LIN {X 0,Y 252.617,Z 375.024,A -85,B 0,C 180,E1 -18754.516,E2 -18754.516} C_VEL
LIN {X 0,Y 250.193,Z 375.321,A -85,B 0,C 180,E1 -18756.259,E2 -18756.259} C_VEL
LIN {X 0,Y 249.15,Z 375.448,A -85,B 0,C 180,E1 -18757.61,E2 -18757.61} C_VEL
LIN {X 0,Y 249.065,Z 375.457,A -85,B 0,C 180,E1 -18758.068,E2 -18758.068} C_VEL
LIN {X 0,Y 249.093,Z 375.454,A -85,B 0,C 180,E1 -18760.461,E2 -18760.461} C_VEL
LIN {X 0,Y 249.089,Z 375.456,A -85,B 0,C 180,E1 -18762.815,E2 -18762.815} C_VEL
LIN {X 0,Y 249.094,Z 375.457,A -85,B 0,C 180,E1 -18767.382,E2 -18767.382} C_VEL
LIN {X 0,Y 249.049,Z 375.461,A -85,B 0,C 180,E1 -18771.626,E2 -18771.626} C_VEL
LIN {X 0,Y 249.193,Z 375.539,A -85,B 0,C 180,E1 -18775.523,E2 -18775.523} C_VEL
LIN {X 0,Y 252.491,Z 392.1,A -85,B 0,C 180,E1 -18780.852,E2 -18780.852} C_VEL
LIN {X 0,Y 253.054,Z 396.272,A -85,B 0,C 180,E1 -18782.147,E2 -18782.147} C_VEL
LIN {X 0,Y 251.958,Z 403.5,A -85,B 0,C 180,E1 -18784.275,E2 -18784.275} C_VEL
LIN {X 0,Y 252.886,Z 424.337,A -85,B 0,C 180,E1 -18785.283,E2 -18785.283} C_VEL
LIN {X 0,Y 255.604,Z 456.086,A -85,B 0,C 180,E1 -18786.853,E2 -18786.853} C_VEL
LIN {X 0,Y 253.392,Z 514.144,A -85,B 0,C 180,E1 -18789.558,E2 -18789.558} C_VEL
LIN {X 0,Y 252.579,Z 527.545,A -85,B 0,C 180,E1 -18790.496,E2 -18790.496} C_VEL
LIN {X 0,Y 251.524,Z 541.094,A -85,B 0,C 180,E1 -18791.809,E2 -18791.809} C_VEL
LIN {X 0,Y 250.583,Z 553.006,A -85,B 0,C 180,E1 -18793.298,E2 -18793.298} C_VEL
LIN {X 0,Y 249.728,Z 563.328,A -85,B 0,C 180,E1 -18794.913,E2 -18794.913} C_VEL
LIN {X 0,Y 248.987,Z 573.942,A -85,B 0,C 180,E1 -18796.951,E2 -18796.951} C_VEL
LIN {X 0,Y 248.46,Z 582.589,A -85,B 0,C 180,E1 -18798.995,E2 -18798.995} C_VEL
LIN {X 0,Y 248.115,Z 590.984,A -85,B 0,C 180,E1 -18801.45,E2 -18801.45} C_VEL
LIN {X 0,Y 248.097,Z 596.674,A -85,B 0,C 180,E1 -18803.496,E2 -18803.496} C_VEL
LIN {X 0,Y 248.11,Z 602.079,A -85,B 0,C 180,E1 -18805.941,E2 -18805.941} C_VEL
LIN {X 0,Y 248.161,Z 606.143,A -85,B 0,C 180,E1 -18808.379,E2 -18808.379} C_VEL
LIN {X 0,Y 248.142,Z 608.182,A -85,B 0,C 180,E1 -18810.002,E2 -18810.002} C_VEL
LIN {X 0,Y 247.812,Z 609.634,A -85,B 0,C 180,E1 -18811.627,E2 -18811.627} C_VEL
LIN {X 0,Y 247.537,Z 610.654,A -85,B 0,C 180,E1 -18813.257,E2 -18813.257} C_VEL
LIN {X 0,Y 247.286,Z 611.402,A -85,B 0,C 180,E1 -18815.888,E2 -18815.888} C_VEL
LIN {X 0,Y 247.279,Z 611.195,A -85,B 0,C 180,E1 -18818.172,E2 -18818.172} C_VEL
LIN {X 0,Y 247.949,Z 609.525,A -85,B 0,C 180,E1 -18821.446,E2 -18821.446} C_VEL
LIN {X 0,Y 248.585,Z 608.119,A -85,B 0,C 180,E1 -18823.074,E2 -18823.074} C_VEL
LIN {X 0,Y 250.166,Z 605.234,A -85,B 0,C 180,E1 -18825.481,E2 -18825.481} C_VEL
LIN {X 0,Y 252.071,Z 601.416,A -85,B 0,C 180,E1 -18827.862,E2 -18827.862} C_VEL
LIN {X 0,Y 254.472,Z 596.794,A -85,B 0,C 180,E1 -18830.113,E2 -18830.113} C_VEL
LIN {X 0,Y 258.315,Z 589.612,A -85,B 0,C 180,E1 -18832.813,E2 -18832.813} C_VEL
LIN {X 0,Y 262.794,Z 580.873,A -85,B 0,C 180,E1 -18835.336,E2 -18835.336} C_VEL
LIN {X 0,Y 267.178,Z 571.753,A -85,B 0,C 180,E1 -18837.41,E2 -18837.41} C_VEL
LIN {X 0,Y 271.297,Z 562.717,A -85,B 0,C 180,E1 -18839.061,E2 -18839.061} C_VEL
LIN {X 0,Y 275.703,Z 552.071,A -85,B 0,C 180,E1 -18840.654,E2 -18840.654} C_VEL
LIN {X 0,Y 280.786,Z 538.915,A -85,B 0,C 180,E1 -18842.134,E2 -18842.134} C_VEL
LIN {X 0,Y 285.07,Z 525.941,A -85,B 0,C 180,E1 -18843.269,E2 -18843.269} C_VEL
LIN {X 0,Y 289,Z 511.6,A -85,B 0,C 180,E1 -18844.243,E2 -18844.243} C_VEL
LIN {X 0,Y 292.448,Z 494.65,A -85,B 0,C 180,E1 -18845.109,E2 -18845.109} C_VEL
LIN {X 0,Y 297.197,Z 467.184,A -85,B 0,C 180,E1 -18846.361,E2 -18846.361} C_VEL
LIN {X 0,Y 297.851,Z 457.621,A -85,B 0,C 180,E1 -18847.315,E2 -18847.315} C_VEL
LIN {X 0,Y 297.997,Z 452.789,A -85,B 0,C 180,E1 -18847.929,E2 -18847.929} C_VEL
LIN {X 0,Y 296.629,Z 446.766,A -85,B 0,C 180,E1 -18849.823,E2 -18849.823} C_VEL
LIN {X 0,Y 295.412,Z 441.538,A -85,B 0,C 180,E1 -18852.263,E2 -18852.263} C_VEL
LIN {X 0,Y 294.804,Z 438.826,A -85,B 0,C 180,E1 -18854.79,E2 -18854.79} C_VEL
LIN {X 0,Y 295.112,Z 437.625,A -85,B 0,C 180,E1 -18856.988,E2 -18856.988} C_VEL
LIN {X 0,Y 295.976,Z 437.721,A -85,B 0,C 180,E1 -18858.968,E2 -18858.968} C_VEL
LIN {X 0,Y 297.649,Z 439.646,A -85,B 0,C 180,E1 -18861.321,E2 -18861.321} C_VEL
LIN {X 0,Y 299.387,Z 442.577,A -85,B 0,C 180,E1 -18863.094,E2 -18863.094} C_VEL
LIN {X 0,Y 300.465,Z 444.609,A -85,B 0,C 180,E1 -18864.024,E2 -18864.024} C_VEL
LIN {X 0,Y 293.198,Z 484.481,A -85,B 0,C 180,E1 -18865.871,E2 -18865.871} C_VEL
LIN {X 0,Y 290.285,Z 498.234,A -85,B 0,C 180,E1 -18866.786,E2 -18866.786} C_VEL
LIN {X 0,Y 287.106,Z 510.262,A -85,B 0,C 180,E1 -18867.831,E2 -18867.831} C_VEL
LIN {X 0,Y 282.774,Z 523.775,A -85,B 0,C 180,E1 -18869.369,E2 -18869.369} C_VEL
LIN {X 0,Y 278.638,Z 534.629,A -85,B 0,C 180,E1 -18870.952,E2 -18870.952} C_VEL
LIN {X 0,Y 273.95,Z 545.313,A -85,B 0,C 180,E1 -18872.911,E2 -18872.911} C_VEL
LIN {X 0,Y 269.585,Z 553.981,A -85,B 0,C 180,E1 -18874.936,E2 -18874.936} C_VEL
LIN {X 0,Y 265.689,Z 561.042,A -85,B 0,C 180,E1 -18877.035,E2 -18877.035} C_VEL
LIN {X 0,Y 261.627,Z 567.566,A -85,B 0,C 180,E1 -18879.56,E2 -18879.56} C_VEL
LIN {X 0,Y 258.489,Z 571.94,A -85,B 0,C 180,E1 -18881.78,E2 -18881.78} C_VEL
LIN {X 0,Y 255.829,Z 575.254,A -85,B 0,C 180,E1 -18884.055,E2 -18884.055} C_VEL
LIN {X 0,Y 252.829,Z 578.178,A -85,B 0,C 180,E1 -18887.151,E2 -18887.151} C_VEL
LIN {X 0,Y 251.574,Z 579.01,A -85,B 0,C 180,E1 -18888.723,E2 -18888.723} C_VEL
LIN {X 0,Y 250.49,Z 579.42,A -85,B 0,C 180,E1 -18890.308,E2 -18890.308} C_VEL
LIN {X 0,Y 249.649,Z 579.428,A -85,B 0,C 180,E1 -18891.908,E2 -18891.908} C_VEL
LIN {X 0,Y 249.079,Z 579.037,A -85,B 0,C 180,E1 -18893.519,E2 -18893.519} C_VEL
LIN {X 0,Y 248.577,Z 578.237,A -85,B 0,C 180,E1 -18895.134,E2 -18895.134} C_VEL
LIN {X 0,Y 248.045,Z 577.007,A -85,B 0,C 180,E1 -18896.751,E2 -18896.751} C_VEL
LIN {X 0,Y 247.507,Z 574.382,A -85,B 0,C 180,E1 -18899.186,E2 -18899.186} C_VEL
LIN {X 0,Y 247.375,Z 570.743,A -85,B 0,C 180,E1 -18901.628,E2 -18901.628} C_VEL
LIN {X 0,Y 247.57,Z 565.989,A -85,B 0,C 180,E1 -18904.07,E2 -18904.07} C_VEL
LIN {X 0,Y 247.729,Z 559.198,A -85,B 0,C 180,E1 -18906.801,E2 -18906.801} C_VEL
LIN {X 0,Y 248.148,Z 552.516,A -85,B 0,C 180,E1 -18908.961,E2 -18908.961} C_VEL
LIN {X 0,Y 248.804,Z 543.249,A -85,B 0,C 180,E1 -18911.404,E2 -18911.404} C_VEL
LIN {X 0,Y 249.629,Z 532.822,A -85,B 0,C 180,E1 -18913.638,E2 -18913.638} C_VEL
LIN {X 0,Y 250.547,Z 522.317,A -85,B 0,C 180,E1 -18915.455,E2 -18915.455} C_VEL
LIN {X 0,Y 251.572,Z 509.36,A -85,B 0,C 180,E1 -18917.267,E2 -18917.267} C_VEL
LIN {X 0,Y 252.418,Z 495.882,A -85,B 0,C 180,E1 -18918.726,E2 -18918.726} C_VEL
LIN {X 0,Y 253.216,Z 482.499,A -85,B 0,C 180,E1 -18919.824,E2 -18919.824} C_VEL
LIN {X 0,Y 253.806,Z 467.784,A -85,B 0,C 180,E1 -18920.674,E2 -18920.674} C_VEL
LIN {X 0,Y 256.435,Z 400.26,A -85,B 0,C 180,E1 -18923.69,E2 -18923.69} C_VEL
LIN {X 0,Y 249.152,Z 375.446,A -85,B 0,C 180,E1 -18925.17,E2 -18925.17} C_VEL
LIN {X 0,Y 249.09,Z 375.455,A -85,B 0,C 180,E1 -18928.993,E2 -18928.993} C_VEL
LIN {X 0,Y 249.039,Z 375.462,A -85,B 0,C 180,E1 -18932.424,E2 -18932.424} C_VEL
LIN {X 0,Y 249.064,Z 375.463,A -85,B 0,C 180,E1 -18936.34,E2 -18936.34} C_VEL
LIN {X 0,Y 249.011,Z 375.465,A -85,B 0,C 180,E1 -18940.477,E2 -18940.477} C_VEL
LIN {X 0,Y 249.007,Z 375.466,A -85,B 0,C 180,E1 -18944.878,E2 -18944.878} C_VEL
LIN {X 0,Y 249.021,Z 375.463,A -85,B 0,C 180,E1 -18947.362,E2 -18947.362} C_VEL
LIN {X 0,Y 249.053,Z 375.462,A -85,B 0,C 180,E1 -18952.197,E2 -18952.197} C_VEL
LIN {X 0,Y 249.063,Z 375.459,A -85,B 0,C 180,E1 -18955.64,E2 -18955.64} C_VEL
LIN {X 0,Y 249.055,Z 375.457,A -85,B 0,C 180,E1 -18959.472,E2 -18959.472} C_VEL
LIN {X 0,Y 249.076,Z 375.457,A -85,B 0,C 180,E1 -18963.161,E2 -18963.161} C_VEL
LIN {X 0,Y 249.083,Z 375.455,A -85,B 0,C 180,E1 -18966.731,E2 -18966.731} C_VEL
LIN {X 0,Y 249.115,Z 375.455,A -85,B 0,C 180,E1 -18970.21,E2 -18970.21} C_VEL
LIN {X 0,Y 249.245,Z 375.437,A -85,B 0,C 180,E1 -18973.62,E2 -18973.62} C_VEL
LIN {X 0,Y 249.247,Z 375.436,A -85,B 0,C 180,E1 -18978.615,E2 -18978.615} C_VEL
LIN {X 0,Y 249.457,Z 375.413,A -85,B 0,C 180,E1 -18981.9,E2 -18981.9} C_VEL
LIN {X 0,Y 249.3,Z 375.427,A -85,B 0,C 180,E1 -18985.147,E2 -18985.147} C_VEL
LIN {X 0,Y 249.678,Z 375.383,A -85,B 0,C 180,E1 -18988.385,E2 -18988.385} C_VEL
LIN {X 0,Y 249.678,Z 375.383,A -85,B 0,C 180,E1 -18991.611,E2 -18991.611} C_VEL
LIN {X 0,Y 249.463,Z 375.409,A -85,B 0,C 180,E1 -18996.468,E2 -18996.468} C_VEL
LIN {X 0,Y 249.424,Z 375.416,A -85,B 0,C 180,E1 -18999.731,E2 -18999.731} C_VEL
LIN {X 0,Y 249.205,Z 375.44,A -85,B 0,C 180,E1 -19004.701,E2 -19004.701} C_VEL
LIN {X 0,Y 249.138,Z 375.452,A -85,B 0,C 180,E1 -19008.075,E2 -19008.075} C_VEL
LIN {X 0,Y 249.085,Z 375.456,A -85,B 0,C 180,E1 -19011.516,E2 -19011.516} C_VEL
LIN {X 0,Y 249.128,Z 375.452,A -85,B 0,C 180,E1 -19015.48,E2 -19015.48} C_VEL
LIN {X 0,Y 249.077,Z 375.456,A -85,B 0,C 180,E1 -19018.99,E2 -19018.99} C_VEL
LIN {X 0,Y 249.032,Z 375.462,A -85,B 0,C 180,E1 -19022.423,E2 -19022.423} C_VEL
LIN {X 0,Y 249.071,Z 375.458,A -85,B 0,C 180,E1 -19026.336,E2 -19026.336} C_VEL
LIN {X 0,Y 249.076,Z 375.456,A -85,B 0,C 180,E1 -19030.461,E2 -19030.461} C_VEL
LIN {X 0,Y 249.082,Z 375.456,A -85,B 0,C 180,E1 -19032.81,E2 -19032.81} C_VEL
LIN {X 0,Y 249.093,Z 375.455,A -85,B 0,C 180,E1 -19037.379,E2 -19037.379} C_VEL
LIN {X 0,Y 249.046,Z 375.464,A -85,B 0,C 180,E1 -19041.623,E2 -19041.623} C_VEL
LIN {X 0,Y 249.054,Z 375.462,A -85,B 0,C 180,E1 -19045.641,E2 -19045.641} C_VEL
LIN {X 0,Y 249.045,Z 375.462,A -85,B 0,C 180,E1 -19049.472,E2 -19049.472} C_VEL
LIN {X 0,Y 249.068,Z 375.459,A -85,B 0,C 180,E1 -19053.162,E2 -19053.162} C_VEL
LIN {X 0,Y 249.071,Z 375.455,A -85,B 0,C 180,E1 -19056.732,E2 -19056.732} C_VEL
LIN {X 0,Y 249.102,Z 375.454,A -85,B 0,C 180,E1 -19060.211,E2 -19060.211} C_VEL
LIN {X 0,Y 249.233,Z 375.439,A -85,B 0,C 180,E1 -19063.621,E2 -19063.621} C_VEL
LIN {X 0,Y 249.244,Z 375.436,A -85,B 0,C 180,E1 -19068.616,E2 -19068.616} C_VEL
LIN {X 0,Y 249.475,Z 375.407,A -85,B 0,C 180,E1 -19071.903,E2 -19071.903} C_VEL
LIN {X 0,Y 249.433,Z 375.412,A -85,B 0,C 180,E1 -19076.77,E2 -19076.77} C_VEL
LIN {X 0,Y 249.727,Z 375.376,A -85,B 0,C 180,E1 -19080,E2 -19080} C_VEL
LIN {X 0,Y 249.431,Z 375.413,A -85,B 0,C 180,E1 -19083.231,E2 -19083.231} C_VEL
LIN {X 0,Y 249.476,Z 375.407,A -85,B 0,C 180,E1 -19088.098,E2 -19088.098} C_VEL
LIN {X 0,Y 249.245,Z 375.437,A -85,B 0,C 180,E1 -19091.384,E2 -19091.384} C_VEL
LIN {X 0,Y 249.234,Z 375.437,A -85,B 0,C 180,E1 -19096.379,E2 -19096.379} C_VEL
LIN {X 0,Y 249.079,Z 375.459,A -85,B 0,C 180,E1 -19101.519,E2 -19101.519} C_VEL
LIN {X 0,Y 249.122,Z 375.454,A -85,B 0,C 180,E1 -19105.483,E2 -19105.483} C_VEL
LIN {X 0,Y 249.065,Z 375.457,A -85,B 0,C 180,E1 -19108.99,E2 -19108.99} C_VEL
LIN {X 0,Y 249.029,Z 375.463,A -85,B 0,C 180,E1 -19112.426,E2 -19112.426} C_VEL
LIN {X 0,Y 249.069,Z 375.456,A -85,B 0,C 180,E1 -19116.339,E2 -19116.339} C_VEL
LIN {X 0,Y 249.065,Z 375.457,A -85,B 0,C 180,E1 -19118.068,E2 -19118.068} C_VEL
LIN {X 0,Y 248.389,Z 375.545,A -85,B 0,C 180,E1 -19119.418,E2 -19119.418} C_VEL
LIN {X 0,Y 245.511,Z 375.903,A -85,B 0,C 180,E1 -19121.617,E2 -19121.617} C_VEL
LIN {X 0,Y 243.082,Z 376.206,A -85,B 0,C 180,E1 -19123.409,E2 -19123.409} C_VEL
LIN {X 0,Y 242.058,Z 376.331,A -85,B 0,C 180,E1 -19124.8,E2 -19124.8} C_VEL
LIN {X 0,Y 241.985,Z 376.336,A -85,B 0,C 180,E1 -19125.271,E2 -19125.271} C_VEL
LIN {X 0,Y 242.006,Z 376.339,A -85,B 0,C 180,E1 -19129.031,E2 -19129.031} C_VEL
LIN {X 0,Y 242.012,Z 376.336,A -85,B 0,C 180,E1 -19132.425,E2 -19132.425} C_VEL
LIN {X 0,Y 242.159,Z 376.504,A -85,B 0,C 180,E1 -19135.409,E2 -19135.409} C_VEL
LIN {X 0,Y 245.444,Z 392.998,A -85,B 0,C 180,E1 -19140.874,E2 -19140.874} C_VEL
LIN {X 0,Y 246.019,Z 395.864,A -85,B 0,C 180,E1 -19141.796,E2 -19141.796} C_VEL
LIN {X 0,Y 244.986,Z 402.846,A -85,B 0,C 180,E1 -19143.945,E2 -19143.945} C_VEL
LIN {X 0,Y 245.82,Z 424.179,A -85,B 0,C 180,E1 -19145.029,E2 -19145.029} C_VEL
LIN {X 0,Y 248.539,Z 456.485,A -85,B 0,C 180,E1 -19146.681,E2 -19146.681} C_VEL
LIN {X 0,Y 246.337,Z 513.372,A -85,B 0,C 180,E1 -19149.437,E2 -19149.437} C_VEL
LIN {X 0,Y 245.574,Z 526.114,A -85,B 0,C 180,E1 -19150.353,E2 -19150.353} C_VEL
LIN {X 0,Y 244.596,Z 538.728,A -85,B 0,C 180,E1 -19151.577,E2 -19151.577} C_VEL
LIN {X 0,Y 243.581,Z 551.828,A -85,B 0,C 180,E1 -19153.232,E2 -19153.232} C_VEL
LIN {X 0,Y 242.707,Z 562.251,A -85,B 0,C 180,E1 -19154.896,E2 -19154.896} C_VEL
LIN {X 0,Y 241.955,Z 572.94,A -85,B 0,C 180,E1 -19156.993,E2 -19156.993} C_VEL
LIN {X 0,Y 241.439,Z 581.655,A -85,B 0,C 180,E1 -19159.096,E2 -19159.096} C_VEL
LIN {X 0,Y 241.112,Z 590.081,A -85,B 0,C 180,E1 -19161.622,E2 -19161.622} C_VEL
LIN {X 0,Y 241.112,Z 596.823,A -85,B 0,C 180,E1 -19164.147,E2 -19164.147} C_VEL
LIN {X 0,Y 241.115,Z 602.029,A -85,B 0,C 180,E1 -19166.66,E2 -19166.66} C_VEL
LIN {X 0,Y 241.167,Z 605.897,A -85,B 0,C 180,E1 -19169.167,E2 -19169.167} C_VEL
LIN {X 0,Y 240.793,Z 608.515,A -85,B 0,C 180,E1 -19171.674,E2 -19171.674} C_VEL
LIN {X 0,Y 240.494,Z 609.654,A -85,B 0,C 180,E1 -19173.353,E2 -19173.353} C_VEL
LIN {X 0,Y 240.23,Z 610.594,A -85,B 0,C 180,E1 -19175.909,E2 -19175.909} C_VEL
LIN {X 0,Y 240.232,Z 610.572,A -85,B 0,C 180,E1 -19178.413,E2 -19178.413} C_VEL
LIN {X 0,Y 240.48,Z 610.095,A -85,B 0,C 180,E1 -19180.101,E2 -19180.101} C_VEL
LIN {X 0,Y 241.647,Z 607.937,A -85,B 0,C 180,E1 -19183.456,E2 -19183.456} C_VEL
LIN {X 0,Y 243.954,Z 604.238,A -85,B 0,C 180,E1 -19186.745,E2 -19186.745} C_VEL
LIN {X 0,Y 246.1,Z 600.387,A -85,B 0,C 180,E1 -19189.174,E2 -19189.174} C_VEL
LIN {X 0,Y 249.066,Z 595.535,A -85,B 0,C 180,E1 -19191.522,E2 -19191.522} C_VEL
LIN {X 0,Y 252.521,Z 589.616,A -85,B 0,C 180,E1 -19193.802,E2 -19193.802} C_VEL
LIN {X 0,Y 257.239,Z 581.183,A -85,B 0,C 180,E1 -19196.359,E2 -19196.359} C_VEL
LIN {X 0,Y 261.893,Z 572.344,A -85,B 0,C 180,E1 -19198.448,E2 -19198.448} C_VEL
LIN {X 0,Y 267.118,Z 561.712,A -85,B 0,C 180,E1 -19200.431,E2 -19200.431} C_VEL
LIN {X 0,Y 271.888,Z 551.1,A -85,B 0,C 180,E1 -19202.001,E2 -19202.001} C_VEL
LIN {X 0,Y 277.23,Z 538.071,A -85,B 0,C 180,E1 -19203.463,E2 -19203.463} C_VEL
LIN {X 0,Y 281.752,Z 525.166,A -85,B 0,C 180,E1 -19204.59,E2 -19204.59} C_VEL
LIN {X 0,Y 286.049,Z 510.245,A -85,B 0,C 180,E1 -19205.597,E2 -19205.597} C_VEL
LIN {X 0,Y 289.59,Z 494.129,A -85,B 0,C 180,E1 -19206.413,E2 -19206.413} C_VEL
LIN {X 0,Y 294.264,Z 468.85,A -85,B 0,C 180,E1 -19207.571,E2 -19207.571} C_VEL
LIN {X 0,Y 295.084,Z 459.535,A -85,B 0,C 180,E1 -19208.557,E2 -19208.557} C_VEL
LIN {X 0,Y 295.153,Z 457.377,A -85,B 0,C 180,E1 -19208.873,E2 -19208.873} C_VEL
LIN {X 0,Y 294.254,Z 452.71,A -85,B 0,C 180,E1 -19210.44,E2 -19210.44} C_VEL
LIN {X 0,Y 293.345,Z 447.937,A -85,B 0,C 180,E1 -19212.734,E2 -19212.734} C_VEL
LIN {X 0,Y 292.987,Z 445.294,A -85,B 0,C 180,E1 -19215.375,E2 -19215.375} C_VEL
LIN {X 0,Y 293.243,Z 444.54,A -85,B 0,C 180,E1 -19216.832,E2 -19216.832} C_VEL
LIN {X 0,Y 294.16,Z 444.64,A -85,B 0,C 180,E1 -19219.006,E2 -19219.006} C_VEL
LIN {X 0,Y 295.622,Z 446.463,A -85,B 0,C 180,E1 -19221.145,E2 -19221.145} C_VEL
LIN {X 0,Y 297.241,Z 449.345,A -85,B 0,C 180,E1 -19222.901,E2 -19222.901} C_VEL
LIN {X 0,Y 289.709,Z 488.112,A -85,B 0,C 180,E1 -19224.766,E2 -19224.766} C_VEL
LIN {X 0,Y 286.648,Z 501.036,A -85,B 0,C 180,E1 -19225.673,E2 -19225.673} C_VEL
LIN {X 0,Y 282.835,Z 513.919,A -85,B 0,C 180,E1 -19226.861,E2 -19226.861} C_VEL
LIN {X 0,Y 278.725,Z 525.572,A -85,B 0,C 180,E1 -19228.24,E2 -19228.24} C_VEL
LIN {X 0,Y 273.913,Z 537.133,A -85,B 0,C 180,E1 -19229.978,E2 -19229.978} C_VEL
LIN {X 0,Y 268.966,Z 547.375,A -85,B 0,C 180,E1 -19231.944,E2 -19231.944} C_VEL
LIN {X 0,Y 264.338,Z 555.79,A -85,B 0,C 180,E1 -19233.979,E2 -19233.979} C_VEL
LIN {X 0,Y 260.171,Z 562.604,A -85,B 0,C 180,E1 -19236.096,E2 -19236.096} C_VEL
LIN {X 0,Y 256.415,Z 568.11,A -85,B 0,C 180,E1 -19238.283,E2 -19238.283} C_VEL
LIN {X 0,Y 253.046,Z 572.496,A -85,B 0,C 180,E1 -19240.532,E2 -19240.532} C_VEL
LIN {X 0,Y 249.99,Z 575.942,A -85,B 0,C 180,E1 -19242.915,E2 -19242.915} C_VEL
LIN {X 0,Y 247.564,Z 578.23,A -85,B 0,C 180,E1 -19245.197,E2 -19245.197} C_VEL
LIN {X 0,Y 244.69,Z 579.952,A -85,B 0,C 180,E1 -19248.401,E2 -19248.401} C_VEL
LIN {X 0,Y 243.539,Z 580.227,A -85,B 0,C 180,E1 -19250.029,E2 -19250.029} C_VEL
LIN {X 0,Y 242.649,Z 580.085,A -85,B 0,C 180,E1 -19251.673,E2 -19251.673} C_VEL
LIN {X 0,Y 241.507,Z 578.539,A -85,B 0,C 180,E1 -19254.991,E2 -19254.991} C_VEL
LIN {X 0,Y 240.961,Z 577.184,A -85,B 0,C 180,E1 -19256.656,E2 -19256.656} C_VEL
LIN {X 0,Y 240.419,Z 574.323,A -85,B 0,C 180,E1 -19259.162,E2 -19259.162} C_VEL
LIN {X 0,Y 240.296,Z 570.436,A -85,B 0,C 180,E1 -19261.676,E2 -19261.676} C_VEL
LIN {X 0,Y 240.504,Z 565.439,A -85,B 0,C 180,E1 -19264.189,E2 -19264.189} C_VEL
LIN {X 0,Y 240.648,Z 558.892,A -85,B 0,C 180,E1 -19266.793,E2 -19266.793} C_VEL
LIN {X 0,Y 241.125,Z 551.302,A -85,B 0,C 180,E1 -19269.225,E2 -19269.225} C_VEL
LIN {X 0,Y 241.823,Z 541.678,A -85,B 0,C 180,E1 -19271.738,E2 -19271.738} C_VEL
LIN {X 0,Y 242.735,Z 530.669,A -85,B 0,C 180,E1 -19274.033,E2 -19274.033} C_VEL
LIN {X 0,Y 243.651,Z 519.657,A -85,B 0,C 180,E1 -19275.904,E2 -19275.904} C_VEL
LIN {X 0,Y 244.58,Z 507.492,A -85,B 0,C 180,E1 -19277.561,E2 -19277.561} C_VEL
LIN {X 0,Y 245.457,Z 493.991,A -85,B 0,C 180,E1 -19279.008,E2 -19279.008} C_VEL
LIN {X 0,Y 246.327,Z 479.034,A -85,B 0,C 180,E1 -19280.185,E2 -19280.185} C_VEL
LIN {X 0,Y 247.021,Z 460.314,A -85,B 0,C 180,E1 -19281.16,E2 -19281.16} C_VEL
LIN {X 0,Y 249.366,Z 401.443,A -85,B 0,C 180,E1 -19283.907,E2 -19283.907} C_VEL
LIN {X 0,Y 242.104,Z 376.324,A -85,B 0,C 180,E1 -19285.457,E2 -19285.457} C_VEL
LIN {X 0,Y 242.036,Z 376.334,A -85,B 0,C 180,E1 -19289.579,E2 -19289.579} C_VEL
LIN {X 0,Y 241.994,Z 376.336,A -85,B 0,C 180,E1 -19293.49,E2 -19293.49} C_VEL
LIN {X 0,Y 241.997,Z 376.339,A -85,B 0,C 180,E1 -19297.58,E2 -19297.58} C_VEL
LIN {X 0,Y 241.943,Z 376.345,A -85,B 0,C 180,E1 -19301.921,E2 -19301.921} C_VEL
LIN {X 0,Y 241.939,Z 376.348,A -85,B 0,C 180,E1 -19306.57,E2 -19306.57} C_VEL
LIN {X 0,Y 241.962,Z 376.344,A -85,B 0,C 180,E1 -19310.28,E2 -19310.28} C_VEL
LIN {X 0,Y 242.041,Z 376.335,A -85,B 0,C 180,E1 -19314.496,E2 -19314.496} C_VEL
LIN {X 0,Y 241.979,Z 376.34,A -85,B 0,C 180,E1 -19318.479,E2 -19318.479} C_VEL
LIN {X 0,Y 242.011,Z 376.34,A -85,B 0,C 180,E1 -19322.311,E2 -19322.311} C_VEL
LIN {X 0,Y 242.061,Z 376.334,A -85,B 0,C 180,E1 -19326.014,E2 -19326.014} C_VEL
LIN {X 0,Y 242.041,Z 376.332,A -85,B 0,C 180,E1 -19329.606,E2 -19329.606} C_VEL
LIN {X 0,Y 242.166,Z 376.318,A -85,B 0,C 180,E1 -19333.277,E2 -19333.277} C_VEL
LIN {X 0,Y 242.184,Z 376.317,A -85,B 0,C 180,E1 -19338.278,E2 -19338.278} C_VEL
LIN {X 0,Y 242.403,Z 376.29,A -85,B 0,C 180,E1 -19341.663,E2 -19341.663} C_VEL
LIN {X 0,Y 242.261,Z 376.303,A -85,B 0,C 180,E1 -19345.005,E2 -19345.005} C_VEL
LIN {X 0,Y 242.639,Z 376.261,A -85,B 0,C 180,E1 -19348.338,E2 -19348.338} C_VEL
LIN {X 0,Y 242.638,Z 376.261,A -85,B 0,C 180,E1 -19351.658,E2 -19351.658} C_VEL
LIN {X 0,Y 242.435,Z 376.284,A -85,B 0,C 180,E1 -19356.657,E2 -19356.657} C_VEL
LIN {X 0,Y 242.345,Z 376.298,A -85,B 0,C 180,E1 -19360.018,E2 -19360.018} C_VEL
LIN {X 0,Y 242.166,Z 376.317,A -85,B 0,C 180,E1 -19365.139,E2 -19365.139} C_VEL
LIN {X 0,Y 242.072,Z 376.329,A -85,B 0,C 180,E1 -19368.622,E2 -19368.622} C_VEL
LIN {X 0,Y 242.01,Z 376.337,A -85,B 0,C 180,E1 -19372.178,E2 -19372.178} C_VEL
LIN {X 0,Y 242.063,Z 376.334,A -85,B 0,C 180,E1 -19375.836,E2 -19375.836} C_VEL
LIN {X 0,Y 242.025,Z 376.336,A -85,B 0,C 180,E1 -19379.578,E2 -19379.578} C_VEL
LIN {X 0,Y 241.987,Z 376.341,A -85,B 0,C 180,E1 -19383.489,E2 -19383.489} C_VEL
LIN {X 0,Y 242.008,Z 376.339,A -85,B 0,C 180,E1 -19387.576,E2 -19387.576} C_VEL
LIN {X 0,Y 242.026,Z 376.338,A -85,B 0,C 180,E1 -19391.9,E2 -19391.9} C_VEL
LIN {X 0,Y 242.019,Z 376.335,A -85,B 0,C 180,E1 -19396.547,E2 -19396.547} C_VEL
LIN {X 0,Y 242.004,Z 376.338,A -85,B 0,C 180,E1 -19400.29,E2 -19400.29} C_VEL
LIN {X 0,Y 242.029,Z 376.334,A -85,B 0,C 180,E1 -19404.496,E2 -19404.496} C_VEL
LIN {X 0,Y 241.969,Z 376.341,A -85,B 0,C 180,E1 -19408.479,E2 -19408.479} C_VEL
LIN {X 0,Y 242.004,Z 376.338,A -85,B 0,C 180,E1 -19412.312,E2 -19412.312} C_VEL
LIN {X 0,Y 242.049,Z 376.332,A -85,B 0,C 180,E1 -19416.015,E2 -19416.015} C_VEL
LIN {X 0,Y 242.029,Z 376.339,A -85,B 0,C 180,E1 -19419.607,E2 -19419.607} C_VEL
LIN {X 0,Y 242.154,Z 376.32,A -85,B 0,C 180,E1 -19423.278,E2 -19423.278} C_VEL
LIN {X 0,Y 242.178,Z 376.316,A -85,B 0,C 180,E1 -19428.28,E2 -19428.28} C_VEL
LIN {X 0,Y 242.426,Z 376.287,A -85,B 0,C 180,E1 -19431.666,E2 -19431.666} C_VEL
LIN {X 0,Y 242.254,Z 376.306,A -85,B 0,C 180,E1 -19435.007,E2 -19435.007} C_VEL
LIN {X 0,Y 242.631,Z 376.26,A -85,B 0,C 180,E1 -19438.34,E2 -19438.34} C_VEL
LIN {X 0,Y 242.629,Z 376.26,A -85,B 0,C 180,E1 -19441.66,E2 -19441.66} C_VEL
LIN {X 0,Y 242.427,Z 376.285,A -85,B 0,C 180,E1 -19446.659,E2 -19446.659} C_VEL
LIN {X 0,Y 242.337,Z 376.295,A -85,B 0,C 180,E1 -19450.021,E2 -19450.021} C_VEL
LIN {X 0,Y 242.159,Z 376.321,A -85,B 0,C 180,E1 -19455.142,E2 -19455.142} C_VEL
LIN {X 0,Y 242.065,Z 376.329,A -85,B 0,C 180,E1 -19458.625,E2 -19458.625} C_VEL
LIN {X 0,Y 242.005,Z 376.337,A -85,B 0,C 180,E1 -19462.181,E2 -19462.181} C_VEL
LIN {X 0,Y 242.059,Z 376.331,A -85,B 0,C 180,E1 -19465.839,E2 -19465.839} C_VEL
LIN {X 0,Y 242,Z 376.34,A -85,B 0,C 180,E1 -19469.585,E2 -19469.585} C_VEL
LIN {X 0,Y 241.984,Z 376.343,A -85,B 0,C 180,E1 -19473.492,E2 -19473.492} C_VEL
LIN {X 0,Y 242.014,Z 376.337,A -85,B 0,C 180,E1 -19477.578,E2 -19477.578} C_VEL
LIN {X 0,Y 242.035,Z 376.334,A -85,B 0,C 180,E1 -19481.902,E2 -19481.902} C_VEL
LIN {X 0,Y 241.985,Z 376.336,A -85,B 0,C 180,E1 -19485.271,E2 -19485.271} C_VEL
LIN {X 0,Y 241.333,Z 376.421,A -85,B 0,C 180,E1 -19486.658,E2 -19486.658} C_VEL
LIN {X 0,Y 238.456,Z 376.781,A -85,B 0,C 180,E1 -19488.921,E2 -19488.921} C_VEL
LIN {X 0,Y 236.017,Z 377.085,A -85,B 0,C 180,E1 -19490.764,E2 -19490.764} C_VEL
LIN {X 0,Y 234.997,Z 377.21,A -85,B 0,C 180,E1 -19492.196,E2 -19492.196} C_VEL
LIN {X 0,Y 234.93,Z 377.217,A -85,B 0,C 180,E1 -19492.682,E2 -19492.682} C_VEL
LIN {X 0,Y 235.09,Z 377.29,A -85,B 0,C 180,E1 -19495.263,E2 -19495.263} C_VEL
LIN {X 0,Y 238.422,Z 393.861,A -85,B 0,C 180,E1 -19500.9,E2 -19500.9} C_VEL
LIN {X 0,Y 238.86,Z 397.113,A -85,B 0,C 180,E1 -19501.97,E2 -19501.97} C_VEL
LIN {X 0,Y 237.999,Z 402.42,A -85,B 0,C 180,E1 -19503.652,E2 -19503.652} C_VEL
LIN {X 0,Y 238.662,Z 422.392,A -85,B 0,C 180,E1 -19504.691,E2 -19504.691} C_VEL
LIN {X 0,Y 241.458,Z 457.036,A -85,B 0,C 180,E1 -19506.524,E2 -19506.524} C_VEL
LIN {X 0,Y 239.258,Z 513.103,A -85,B 0,C 180,E1 -19509.363,E2 -19509.363} C_VEL
LIN {X 0,Y 238.496,Z 525.74,A -85,B 0,C 180,E1 -19510.306,E2 -19510.306} C_VEL
LIN {X 0,Y 237.515,Z 538.258,A -85,B 0,C 180,E1 -19511.569,E2 -19511.569} C_VEL
LIN {X 0,Y 236.596,Z 550.537,A -85,B 0,C 180,E1 -19513.167,E2 -19513.167} C_VEL
LIN {X 0,Y 235.712,Z 561.083,A -85,B 0,C 180,E1 -19514.879,E2 -19514.879} C_VEL
LIN {X 0,Y 234.953,Z 571.823,A -85,B 0,C 180,E1 -19517.038,E2 -19517.038} C_VEL
LIN {X 0,Y 234.454,Z 580.635,A -85,B 0,C 180,E1 -19519.204,E2 -19519.204} C_VEL
LIN {X 0,Y 234.148,Z 588.901,A -85,B 0,C 180,E1 -19521.727,E2 -19521.727} C_VEL
LIN {X 0,Y 234.15,Z 595.895,A -85,B 0,C 180,E1 -19524.404,E2 -19524.404} C_VEL
LIN {X 0,Y 234.15,Z 600.345,A -85,B 0,C 180,E1 -19526.56,E2 -19526.56} C_VEL
LIN {X 0,Y 234.194,Z 604.452,A -85,B 0,C 180,E1 -19529.142,E2 -19529.142} C_VEL
LIN {X 0,Y 234.193,Z 605.556,A -85,B 0,C 180,E1 -19530.002,E2 -19530.002} C_VEL
LIN {X 0,Y 233.794,Z 607.279,A -85,B 0,C 180,E1 -19531.725,E2 -19531.725} C_VEL
LIN {X 0,Y 233.49,Z 608.564,A -85,B 0,C 180,E1 -19533.453,E2 -19533.453} C_VEL
LIN {X 0,Y 233.208,Z 609.67,A -85,B 0,C 180,E1 -19536.013,E2 -19536.013} C_VEL
LIN {X 0,Y 233.181,Z 609.893,A -85,B 0,C 180,E1 -19538.669,E2 -19538.669} C_VEL
LIN {X 0,Y 233.967,Z 608.817,A -85,B 0,C 180,E1 -19542.14,E2 -19542.14} C_VEL
LIN {X 0,Y 234.727,Z 607.722,A -85,B 0,C 180,E1 -19543.861,E2 -19543.861} C_VEL
LIN {X 0,Y 235.848,Z 606.254,A -85,B 0,C 180,E1 -19545.558,E2 -19545.558} C_VEL
LIN {X 0,Y 238.587,Z 602.094,A -85,B 0,C 180,E1 -19548.908,E2 -19548.908} C_VEL
LIN {X 0,Y 241.755,Z 597.396,A -85,B 0,C 180,E1 -19551.602,E2 -19551.602} C_VEL
LIN {X 0,Y 244.76,Z 592.751,A -85,B 0,C 180,E1 -19553.705,E2 -19553.705} C_VEL
LIN {X 0,Y 249.559,Z 585.266,A -85,B 0,C 180,E1 -19556.332,E2 -19556.332} C_VEL
LIN {X 0,Y 255.021,Z 576.074,A -85,B 0,C 180,E1 -19558.836,E2 -19558.836} C_VEL
LIN {X 0,Y 260.319,Z 566.447,A -85,B 0,C 180,E1 -19560.863,E2 -19560.863} C_VEL
LIN {X 0,Y 266.127,Z 554.889,A -85,B 0,C 180,E1 -19562.779,E2 -19562.779} C_VEL
LIN {X 0,Y 272.15,Z 541.707,A -85,B 0,C 180,E1 -19564.397,E2 -19564.397} C_VEL
LIN {X 0,Y 277.369,Z 528.402,A -85,B 0,C 180,E1 -19565.648,E2 -19565.648} C_VEL
LIN {X 0,Y 282.207,Z 513.606,A -85,B 0,C 180,E1 -19566.706,E2 -19566.706} C_VEL
LIN {X 0,Y 286.021,Z 498.724,A -85,B 0,C 180,E1 -19567.525,E2 -19567.525} C_VEL
LIN {X 0,Y 291.655,Z 470.421,A -85,B 0,C 180,E1 -19568.837,E2 -19568.837} C_VEL
LIN {X 0,Y 292.514,Z 462.362,A -85,B 0,C 180,E1 -19569.75,E2 -19569.75} C_VEL
LIN {X 0,Y 291.908,Z 458.502,A -85,B 0,C 180,E1 -19571.14,E2 -19571.14} C_VEL
LIN {X 0,Y 291.362,Z 454.431,A -85,B 0,C 180,E1 -19573.145,E2 -19573.145} C_VEL
LIN {X 0,Y 291.189,Z 451.94,A -85,B 0,C 180,E1 -19575.735,E2 -19575.735} C_VEL
LIN {X 0,Y 291.638,Z 451.286,A -85,B 0,C 180,E1 -19577.565,E2 -19577.565} C_VEL
LIN {X 0,Y 292.419,Z 451.651,A -85,B 0,C 180,E1 -19579.203,E2 -19579.203} C_VEL
LIN {X 0,Y 293.536,Z 453.108,A -85,B 0,C 180,E1 -19580.882,E2 -19580.882} C_VEL
LIN {X 0,Y 294.257,Z 454.46,A -85,B 0,C 180,E1 -19581.792,E2 -19581.792} C_VEL
LIN {X 0,Y 287.079,Z 489.119,A -85,B 0,C 180,E1 -19583.473,E2 -19583.473} C_VEL
LIN {X 0,Y 283.717,Z 502.324,A -85,B 0,C 180,E1 -19584.4,E2 -19584.4} C_VEL
LIN {X 0,Y 279.674,Z 514.958,A -85,B 0,C 180,E1 -19585.569,E2 -19585.569} C_VEL
LIN {X 0,Y 274.838,Z 527.573,A -85,B 0,C 180,E1 -19587.085,E2 -19587.085} C_VEL
LIN {X 0,Y 270.223,Z 537.869,A -85,B 0,C 180,E1 -19588.657,E2 -19588.657} C_VEL
LIN {X 0,Y 264.92,Z 548.068,A -85,B 0,C 180,E1 -19590.608,E2 -19590.608} C_VEL
LIN {X 0,Y 259.989,Z 556.418,A -85,B 0,C 180,E1 -19592.642,E2 -19592.642} C_VEL
LIN {X 0,Y 255.475,Z 563.239,A -85,B 0,C 180,E1 -19594.761,E2 -19594.761} C_VEL
LIN {X 0,Y 251.4,Z 568.746,A -85,B 0,C 180,E1 -19596.96,E2 -19596.96} C_VEL
LIN {X 0,Y 247.763,Z 573.128,A -85,B 0,C 180,E1 -19599.233,E2 -19599.233} C_VEL
LIN {X 0,Y 244.476,Z 576.508,A -85,B 0,C 180,E1 -19601.565,E2 -19601.565} C_VEL
LIN {X 0,Y 240.816,Z 579.476,A -85,B 0,C 180,E1 -19604.772,E2 -19604.772} C_VEL
LIN {X 0,Y 237.815,Z 580.882,A -85,B 0,C 180,E1 -19608.061,E2 -19608.061} C_VEL
LIN {X 0,Y 236.586,Z 580.956,A -85,B 0,C 180,E1 -19609.733,E2 -19609.733} C_VEL
LIN {X 0,Y 234.99,Z 579.919,A -85,B 0,C 180,E1 -19613.129,E2 -19613.129} C_VEL
LIN {X 0,Y 234.439,Z 578.815,A -85,B 0,C 180,E1 -19614.84,E2 -19614.84} C_VEL
LIN {X 0,Y 233.881,Z 577.268,A -85,B 0,C 180,E1 -19616.554,E2 -19616.554} C_VEL
LIN {X 0,Y 233.332,Z 574.173,A -85,B 0,C 180,E1 -19619.137,E2 -19619.137} C_VEL
LIN {X 0,Y 233.219,Z 570.032,A -85,B 0,C 180,E1 -19621.727,E2 -19621.727} C_VEL
LIN {X 0,Y 233.437,Z 564.754,A -85,B 0,C 180,E1 -19624.316,E2 -19624.316} C_VEL
LIN {X 0,Y 233.689,Z 556.904,A -85,B 0,C 180,E1 -19627.343,E2 -19627.343} C_VEL
LIN {X 0,Y 234.236,Z 548.431,A -85,B 0,C 180,E1 -19629.934,E2 -19629.934} C_VEL
LIN {X 0,Y 235.003,Z 537.947,A -85,B 0,C 180,E1 -19632.522,E2 -19632.522} C_VEL
LIN {X 0,Y 236.055,Z 525.946,A -85,B 0,C 180,E1 -19634.88,E2 -19634.88} C_VEL
LIN {X 0,Y 237.062,Z 513.695,A -85,B 0,C 180,E1 -19636.801,E2 -19636.801} C_VEL
LIN {X 0,Y 237.85,Z 501.737,A -85,B 0,C 180,E1 -19638.297,E2 -19638.297} C_VEL
LIN {X 0,Y 238.73,Z 488.319,A -85,B 0,C 180,E1 -19639.596,E2 -19639.596} C_VEL
LIN {X 0,Y 239.392,Z 474.547,A -85,B 0,C 180,E1 -19640.58,E2 -19640.58} C_VEL
LIN {X 0,Y 242.351,Z 402.68,A -85,B 0,C 180,E1 -19644.102,E2 -19644.102} C_VEL
LIN {X 0,Y 235.04,Z 377.204,A -85,B 0,C 180,E1 -19645.721,E2 -19645.721} C_VEL
LIN {X 0,Y 234.938,Z 377.219,A -85,B 0,C 180,E1 -19650.567,E2 -19650.567} C_VEL
LIN {X 0,Y 234.948,Z 377.218,A -85,B 0,C 180,E1 -19654.635,E2 -19654.635} C_VEL
LIN {X 0,Y 234.947,Z 377.217,A -85,B 0,C 180,E1 -19658.943,E2 -19658.943} C_VEL
LIN {X 0,Y 234.892,Z 377.222,A -85,B 0,C 180,E1 -19663.485,E2 -19663.485} C_VEL
LIN {X 0,Y 234.892,Z 377.226,A -85,B 0,C 180,E1 -19666.513,E2 -19666.513} C_VEL
LIN {X 0,Y 234.924,Z 377.217,A -85,B 0,C 180,E1 -19671.078,E2 -19671.078} C_VEL
LIN {X 0,Y 234.964,Z 377.215,A -85,B 0,C 180,E1 -19675.366,E2 -19675.366} C_VEL
LIN {X 0,Y 234.972,Z 377.214,A -85,B 0,C 180,E1 -19680.156,E2 -19680.156} C_VEL
LIN {X 0,Y 234.998,Z 377.212,A -85,B 0,C 180,E1 -19683.792,E2 -19683.792} C_VEL
LIN {X 0,Y 235.015,Z 377.206,A -85,B 0,C 180,E1 -19688.968,E2 -19688.968} C_VEL
LIN {X 0,Y 235.1,Z 377.198,A -85,B 0,C 180,E1 -19693.058,E2 -19693.058} C_VEL
LIN {X 0,Y 235.118,Z 377.196,A -85,B 0,C 180,E1 -19697.92,E2 -19697.92} C_VEL
LIN {X 0,Y 235.334,Z 377.169,A -85,B 0,C 180,E1 -19701.411,E2 -19701.411} C_VEL
LIN {X 0,Y 235.376,Z 377.163,A -85,B 0,C 180,E1 -19703.139,E2 -19703.139} C_VEL
LIN {X 0,Y 235.598,Z 377.138,A -85,B 0,C 180,E1 -19708.289,E2 -19708.289} C_VEL
LIN {X 0,Y 235.598,Z 377.138,A -85,B 0,C 180,E1 -19711.707,E2 -19711.707} C_VEL
LIN {X 0,Y 235.407,Z 377.159,A -85,B 0,C 180,E1 -19716.857,E2 -19716.857} C_VEL
LIN {X 0,Y 235.253,Z 377.18,A -85,B 0,C 180,E1 -19720.324,E2 -19720.324} C_VEL
LIN {X 0,Y 235.113,Z 377.197,A -85,B 0,C 180,E1 -19725.604,E2 -19725.604} C_VEL
LIN {X 0,Y 235.007,Z 377.209,A -85,B 0,C 180,E1 -19729.203,E2 -19729.203} C_VEL
LIN {X 0,Y 234.959,Z 377.213,A -85,B 0,C 180,E1 -19732.881,E2 -19732.881} C_VEL
LIN {X 0,Y 234.966,Z 377.215,A -85,B 0,C 180,E1 -19736.655,E2 -19736.655} C_VEL
LIN {X 0,Y 234.928,Z 377.216,A -85,B 0,C 180,E1 -19740.566,E2 -19740.566} C_VEL
LIN {X 0,Y 234.956,Z 377.216,A -85,B 0,C 180,E1 -19744.631,E2 -19744.631} C_VEL
LIN {X 0,Y 234.961,Z 377.213,A -85,B 0,C 180,E1 -19748.95,E2 -19748.95} C_VEL
LIN {X 0,Y 234.987,Z 377.214,A -85,B 0,C 180,E1 -19753.46,E2 -19753.46} C_VEL
LIN {X 0,Y 234.991,Z 377.21,A -85,B 0,C 180,E1 -19756.538,E2 -19756.538} C_VEL
LIN {X 0,Y 234.948,Z 377.217,A -85,B 0,C 180,E1 -19761.085,E2 -19761.085} C_VEL
LIN {X 0,Y 234.953,Z 377.217,A -85,B 0,C 180,E1 -19765.366,E2 -19765.366} C_VEL
LIN {X 0,Y 234.962,Z 377.216,A -85,B 0,C 180,E1 -19770.156,E2 -19770.156} C_VEL
LIN {X 0,Y 234.986,Z 377.213,A -85,B 0,C 180,E1 -19773.793,E2 -19773.793} C_VEL
LIN {X 0,Y 235.003,Z 377.21,A -85,B 0,C 180,E1 -19778.969,E2 -19778.969} C_VEL
LIN {X 0,Y 235.088,Z 377.199,A -85,B 0,C 180,E1 -19783.059,E2 -19783.059} C_VEL
LIN {X 0,Y 235.138,Z 377.195,A -85,B 0,C 180,E1 -19787.923,E2 -19787.923} C_VEL
LIN {X 0,Y 235.381,Z 377.166,A -85,B 0,C 180,E1 -19791.414,E2 -19791.414} C_VEL
LIN {X 0,Y 235.397,Z 377.16,A -85,B 0,C 180,E1 -19793.141,E2 -19793.141} C_VEL
LIN {X 0,Y 235.59,Z 377.137,A -85,B 0,C 180,E1 -19798.291,E2 -19798.291} C_VEL
LIN {X 0,Y 235.589,Z 377.137,A -85,B 0,C 180,E1 -19801.71,E2 -19801.71} C_VEL
LIN {X 0,Y 235.398,Z 377.161,A -85,B 0,C 180,E1 -19806.859,E2 -19806.859} C_VEL
LIN {X 0,Y 235.245,Z 377.177,A -85,B 0,C 180,E1 -19810.326,E2 -19810.326} C_VEL
LIN {X 0,Y 235.106,Z 377.2,A -85,B 0,C 180,E1 -19815.607,E2 -19815.607} C_VEL
LIN {X 0,Y 235.001,Z 377.211,A -85,B 0,C 180,E1 -19819.206,E2 -19819.206} C_VEL
LIN {X 0,Y 234.953,Z 377.217,A -85,B 0,C 180,E1 -19822.884,E2 -19822.884} C_VEL
LIN {X 0,Y 234.96,Z 377.215,A -85,B 0,C 180,E1 -19826.659,E2 -19826.659} C_VEL
LIN {X 0,Y 234.916,Z 377.22,A -85,B 0,C 180,E1 -19830.57,E2 -19830.57} C_VEL
LIN {X 0,Y 234.954,Z 377.216,A -85,B 0,C 180,E1 -19834.634,E2 -19834.634} C_VEL
LIN {X 0,Y 234.991,Z 377.211,A -85,B 0,C 180,E1 -19838.963,E2 -19838.963} C_VEL
LIN {X 0,Y 234.991,Z 377.213,A -85,B 0,C 180,E1 -19843.462,E2 -19843.462} C_VEL
LIN {X 0,Y 234.992,Z 377.208,A -85,B 0,C 180,E1 -19846.541,E2 -19846.541} C_VEL
LIN {X 0,Y 234.966,Z 377.218,A -85,B 0,C 180,E1 -19851.091,E2 -19851.091} C_VEL
LIN {X 0,Y 234.93,Z 377.217,A -85,B 0,C 180,E1 -19852.682,E2 -19852.682} C_VEL
LIN {X 0,Y 234.696,Z 377.573,A -85,B 0,C 180,E1 -19853.626,E2 -19853.626} C_VEL
LIN {X 0,Y 233.653,Z 379.175,A -85,B 0,C 180,E1 -19854.987,E2 -19854.987} C_VEL
LIN {X 0,Y 232.265,Z 381.675,A -85,B 0,C 180,E1 -19856.268,E2 -19856.268} C_VEL
LIN {X 0,Y 230.658,Z 385.965,A -85,B 0,C 180,E1 -19857.93,E2 -19857.93} C_VEL
LIN {X 0,Y 230.332,Z 389.486,A -85,B 0,C 180,E1 -19859.155,E2 -19859.155} C_VEL
LIN {X 0,Y 230.501,Z 390.664,A -85,B 0,C 180,E1 -19859.561,E2 -19859.561} C_VEL
LIN {X 0,Y 231.74,Z 396.542,A -85,B 0,C 180,E1 -19861.581,E2 -19861.581} C_VEL
LIN {X 0,Y 231.028,Z 401.913,A -85,B 0,C 180,E1 -19863.342,E2 -19863.342} C_VEL
LIN {X 0,Y 231.526,Z 421.625,A -85,B 0,C 180,E1 -19864.402,E2 -19864.402} C_VEL
LIN {X 0,Y 234.406,Z 457.297,A -85,B 0,C 180,E1 -19866.362,E2 -19866.362} C_VEL
LIN {X 0,Y 232.209,Z 512.455,A -85,B 0,C 180,E1 -19869.281,E2 -19869.281} C_VEL
LIN {X 0,Y 231.391,Z 525.722,A -85,B 0,C 180,E1 -19870.316,E2 -19870.316} C_VEL
LIN {X 0,Y 230.376,Z 538.794,A -85,B 0,C 180,E1 -19871.706,E2 -19871.706} C_VEL
LIN {X 0,Y 229.462,Z 550.591,A -85,B 0,C 180,E1 -19873.316,E2 -19873.316} C_VEL
LIN {X 0,Y 228.609,Z 560.96,A -85,B 0,C 180,E1 -19875.082,E2 -19875.082} C_VEL
LIN {X 0,Y 227.964,Z 570.625,A -85,B 0,C 180,E1 -19877.087,E2 -19877.087} C_VEL
LIN {X 0,Y 227.479,Z 579.5,A -85,B 0,C 180,E1 -19879.319,E2 -19879.319} C_VEL
LIN {X 0,Y 227.181,Z 587.745,A -85,B 0,C 180,E1 -19881.87,E2 -19881.87} C_VEL
LIN {X 0,Y 227.182,Z 594.908,A -85,B 0,C 180,E1 -19884.677,E2 -19884.677} C_VEL
LIN {X 0,Y 227.221,Z 600.189,A -85,B 0,C 180,E1 -19887.343,E2 -19887.343} C_VEL
LIN {X 0,Y 227.229,Z 604.119,A -85,B 0,C 180,E1 -19890.002,E2 -19890.002} C_VEL
LIN {X 0,Y 226.803,Z 606.007,A -85,B 0,C 180,E1 -19891.778,E2 -19891.778} C_VEL
LIN {X 0,Y 226.481,Z 607.414,A -85,B 0,C 180,E1 -19893.56,E2 -19893.56} C_VEL
LIN {X 0,Y 226.101,Z 608.96,A -85,B 0,C 180,E1 -19897.144,E2 -19897.144} C_VEL
LIN {X 0,Y 226.455,Z 608.972,A -85,B 0,C 180,E1 -19900.734,E2 -19900.734} C_VEL
LIN {X 0,Y 227.826,Z 607.446,A -85,B 0,C 180,E1 -19904.289,E2 -19904.289} C_VEL
LIN {X 0,Y 230.33,Z 604.44,A -85,B 0,C 180,E1 -19907.768,E2 -19907.768} C_VEL
LIN {X 0,Y 233.708,Z 599.928,A -85,B 0,C 180,E1 -19911.155,E2 -19911.155} C_VEL
LIN {X 0,Y 238.345,Z 593.695,A -85,B 0,C 180,E1 -19914.384,E2 -19914.384} C_VEL
LIN {X 0,Y 243.353,Z 586.729,A -85,B 0,C 180,E1 -19917.058,E2 -19917.058} C_VEL
LIN {X 0,Y 249.019,Z 578.116,A -85,B 0,C 180,E1 -19919.599,E2 -19919.599} C_VEL
LIN {X 0,Y 254.469,Z 569.175,A -85,B 0,C 180,E1 -19921.653,E2 -19921.653} C_VEL
LIN {X 0,Y 260.958,Z 557.485,A -85,B 0,C 180,E1 -19923.744,E2 -19923.744} C_VEL
LIN {X 0,Y 267.248,Z 545.058,A -85,B 0,C 180,E1 -19925.39,E2 -19925.39} C_VEL
LIN {X 0,Y 273.291,Z 531.213,A -85,B 0,C 180,E1 -19926.777,E2 -19926.777} C_VEL
LIN {X 0,Y 278.815,Z 516.06,A -85,B 0,C 180,E1 -19927.911,E2 -19927.911} C_VEL
LIN {X 0,Y 282.973,Z 501.641,A -85,B 0,C 180,E1 -19928.748,E2 -19928.748} C_VEL
LIN {X 0,Y 289.307,Z 472.572,A -85,B 0,C 180,E1 -19930.094,E2 -19930.094} C_VEL
LIN {X 0,Y 290.002,Z 467.365,A -85,B 0,C 180,E1 -19930.68,E2 -19930.68} C_VEL
LIN {X 0,Y 289.728,Z 464.756,A -85,B 0,C 180,E1 -19931.632,E2 -19931.632} C_VEL
LIN {X 0,Y 289.373,Z 460.89,A -85,B 0,C 180,E1 -19933.592,E2 -19933.592} C_VEL
LIN {X 0,Y 289.403,Z 458.647,A -85,B 0,C 180,E1 -19936.121,E2 -19936.121} C_VEL
LIN {X 0,Y 289.694,Z 458.189,A -85,B 0,C 180,E1 -19937.212,E2 -19937.212} C_VEL
LIN {X 0,Y 290.432,Z 458.377,A -85,B 0,C 180,E1 -19938.932,E2 -19938.932} C_VEL
LIN {X 0,Y 291.462,Z 459.796,A -85,B 0,C 180,E1 -19940.637,E2 -19940.637} C_VEL
LIN {X 0,Y 291.38,Z 460.373,A -85,B 0,C 180,E1 -19940.705,E2 -19940.705} C_VEL
LIN {X 0,Y 285.128,Z 488.923,A -85,B 0,C 180,E1 -19942.071,E2 -19942.071} C_VEL
LIN {X 0,Y 281.561,Z 502.132,A -85,B 0,C 180,E1 -19942.973,E2 -19942.973} C_VEL
LIN {X 0,Y 277.798,Z 513.495,A -85,B 0,C 180,E1 -19943.97,E2 -19943.97} C_VEL
LIN {X 0,Y 272.651,Z 526.426,A -85,B 0,C 180,E1 -19945.453,E2 -19945.453} C_VEL
LIN {X 0,Y 267.684,Z 536.973,A -85,B 0,C 180,E1 -19946.989,E2 -19946.989} C_VEL
LIN {X 0,Y 262.037,Z 547.408,A -85,B 0,C 180,E1 -19948.916,E2 -19948.916} C_VEL
LIN {X 0,Y 256.69,Z 555.935,A -85,B 0,C 180,E1 -19950.923,E2 -19950.923} C_VEL
LIN {X 0,Y 251.754,Z 562.945,A -85,B 0,C 180,E1 -19953.022,E2 -19953.022} C_VEL
LIN {X 0,Y 246.58,Z 569.479,A -85,B 0,C 180,E1 -19955.589,E2 -19955.589} C_VEL
LIN {X 0,Y 242.634,Z 573.84,A -85,B 0,C 180,E1 -19957.88,E2 -19957.88} C_VEL
LIN {X 0,Y 237.92,Z 578.102,A -85,B 0,C 180,E1 -19961.038,E2 -19961.038} C_VEL
LIN {X 0,Y 235.873,Z 579.621,A -85,B 0,C 180,E1 -19962.665,E2 -19962.665} C_VEL
LIN {X 0,Y 234.082,Z 580.709,A -85,B 0,C 180,E1 -19964.323,E2 -19964.323} C_VEL
LIN {X 0,Y 230.921,Z 581.712,A -85,B 0,C 180,E1 -19967.699,E2 -19967.699} C_VEL
LIN {X 0,Y 229.639,Z 581.638,A -85,B 0,C 180,E1 -19969.419,E2 -19969.419} C_VEL
LIN {X 0,Y 228.655,Z 581.161,A -85,B 0,C 180,E1 -19971.159,E2 -19971.159} C_VEL
LIN {X 0,Y 227.376,Z 578.962,A -85,B 0,C 180,E1 -19974.679,E2 -19974.679} C_VEL
LIN {X 0,Y 226.561,Z 576.264,A -85,B 0,C 180,E1 -19977.333,E2 -19977.333} C_VEL
LIN {X 0,Y 226.179,Z 572.569,A -85,B 0,C 180,E1 -19980,E2 -19980} C_VEL
LIN {X 0,Y 226.196,Z 567.799,A -85,B 0,C 180,E1 -19982.671,E2 -19982.671} C_VEL
LIN {X 0,Y 226.356,Z 561.785,A -85,B 0,C 180,E1 -19985.344,E2 -19985.344} C_VEL
LIN {X 0,Y 226.76,Z 554.375,A -85,B 0,C 180,E1 -19988.017,E2 -19988.017} C_VEL
LIN {X 0,Y 227.358,Z 545.159,A -85,B 0,C 180,E1 -19990.688,E2 -19990.688} C_VEL
LIN {X 0,Y 228.163,Z 534.805,A -85,B 0,C 180,E1 -19993.13,E2 -19993.13} C_VEL
LIN {X 0,Y 229.162,Z 523.187,A -85,B 0,C 180,E1 -19995.338,E2 -19995.338} C_VEL
LIN {X 0,Y 230.122,Z 511.757,A -85,B 0,C 180,E1 -19997.094,E2 -19997.094} C_VEL
LIN {X 0,Y 231.008,Z 498.124,A -85,B 0,C 180,E1 -19998.744,E2 -19998.744} C_VEL
LIN {X 0,Y 231.882,Z 484.252,A -85,B 0,C 180,E1 -20000.017,E2 -20000.017} C_VEL
LIN {X 0,Y 232.549,Z 469.199,A -85,B 0,C 180,E1 -20000.99,E2 -20000.99} C_VEL
LIN {X 0,Y 235.229,Z 403.52,A -85,B 0,C 180,E1 -20004.318,E2 -20004.318} C_VEL
LIN {X 0,Y 228.005,Z 378.081,A -85,B 0,C 180,E1 -20005.97,E2 -20005.97} C_VEL
LIN {X 0,Y 227.915,Z 378.096,A -85,B 0,C 180,E1 -20010.295,E2 -20010.295} C_VEL
LIN {X 0,Y 227.886,Z 378.094,A -85,B 0,C 180,E1 -20013.719,E2 -20013.719} C_VEL
LIN {X 0,Y 227.85,Z 378.104,A -85,B 0,C 180,E1 -20018.09,E2 -20018.09} C_VEL
LIN {X 0,Y 227.816,Z 378.105,A -85,B 0,C 180,E1 -20022.741,E2 -20022.741} C_VEL
LIN {X 0,Y 227.816,Z 378.105,A -85,B 0,C 180,E1 -20027.256,E2 -20027.256} C_VEL
LIN {X 0,Y 227.853,Z 378.1,A -85,B 0,C 180,E1 -20031.908,E2 -20031.908} C_VEL
LIN {X 0,Y 227.893,Z 378.098,A -85,B 0,C 180,E1 -20036.28,E2 -20036.28} C_VEL
LIN {X 0,Y 227.922,Z 378.093,A -85,B 0,C 180,E1 -20040.436,E2 -20040.436} C_VEL
LIN {X 0,Y 227.932,Z 378.092,A -85,B 0,C 180,E1 -20044.424,E2 -20044.424} C_VEL
LIN {X 0,Y 227.966,Z 378.087,A -85,B 0,C 180,E1 -20048.285,E2 -20048.285} C_VEL
LIN {X 0,Y 228.038,Z 378.078,A -85,B 0,C 180,E1 -20052.824,E2 -20052.824} C_VEL
LIN {X 0,Y 228.076,Z 378.07,A -85,B 0,C 180,E1 -20057.541,E2 -20057.541} C_VEL
LIN {X 0,Y 228.27,Z 378.049,A -85,B 0,C 180,E1 -20061.143,E2 -20061.143} C_VEL
LIN {X 0,Y 228.327,Z 378.041,A -85,B 0,C 180,E1 -20062.926,E2 -20062.926} C_VEL
LIN {X 0,Y 228.557,Z 378.015,A -85,B 0,C 180,E1 -20068.236,E2 -20068.236} C_VEL
LIN {X 0,Y 228.557,Z 378.015,A -85,B 0,C 180,E1 -20071.76,E2 -20071.76} C_VEL
LIN {X 0,Y 228.359,Z 378.037,A -85,B 0,C 180,E1 -20077.069,E2 -20077.069} C_VEL
LIN {X 0,Y 228.171,Z 378.06,A -85,B 0,C 180,E1 -20080.648,E2 -20080.648} C_VEL
LIN {X 0,Y 228.056,Z 378.078,A -85,B 0,C 180,E1 -20086.1,E2 -20086.1} C_VEL
LIN {X 0,Y 227.941,Z 378.092,A -85,B 0,C 180,E1 -20089.823,E2 -20089.823} C_VEL
LIN {X 0,Y 227.911,Z 378.093,A -85,B 0,C 180,E1 -20093.63,E2 -20093.63} C_VEL
LIN {X 0,Y 227.882,Z 378.099,A -85,B 0,C 180,E1 -20097.553,E2 -20097.553} C_VEL
LIN {X 0,Y 227.869,Z 378.098,A -85,B 0,C 180,E1 -20101.62,E2 -20101.62} C_VEL
LIN {X 0,Y 227.897,Z 378.098,A -85,B 0,C 180,E1 -20105.866,E2 -20105.866} C_VEL
LIN {X 0,Y 227.896,Z 378.094,A -85,B 0,C 180,E1 -20110.359,E2 -20110.359} C_VEL
LIN {X 0,Y 227.913,Z 378.093,A -85,B 0,C 180,E1 -20114.827,E2 -20114.827} C_VEL
LIN {X 0,Y 227.929,Z 378.092,A -85,B 0,C 180,E1 -20117.73,E2 -20117.73} C_VEL
LIN {X 0,Y 227.864,Z 378.102,A -85,B 0,C 180,E1 -20121.913,E2 -20121.913} C_VEL
LIN {X 0,Y 227.883,Z 378.094,A -85,B 0,C 180,E1 -20126.372,E2 -20126.372} C_VEL
LIN {X 0,Y 227.912,Z 378.093,A -85,B 0,C 180,E1 -20130.437,E2 -20130.437} C_VEL
LIN {X 0,Y 227.921,Z 378.09,A -85,B 0,C 180,E1 -20134.425,E2 -20134.425} C_VEL
LIN {X 0,Y 227.954,Z 378.088,A -85,B 0,C 180,E1 -20138.286,E2 -20138.286} C_VEL
LIN {X 0,Y 228.026,Z 378.078,A -85,B 0,C 180,E1 -20142.825,E2 -20142.825} C_VEL
LIN {X 0,Y 228.086,Z 378.074,A -85,B 0,C 180,E1 -20147.544,E2 -20147.544} C_VEL
LIN {X 0,Y 228.316,Z 378.044,A -85,B 0,C 180,E1 -20151.147,E2 -20151.147} C_VEL
LIN {X 0,Y 228.349,Z 378.037,A -85,B 0,C 180,E1 -20152.929,E2 -20152.929} C_VEL
LIN {X 0,Y 228.549,Z 378.014,A -85,B 0,C 180,E1 -20158.238,E2 -20158.238} C_VEL
LIN {X 0,Y 228.547,Z 378.013,A -85,B 0,C 180,E1 -20161.762,E2 -20161.762} C_VEL
LIN {X 0,Y 228.35,Z 378.04,A -85,B 0,C 180,E1 -20167.072,E2 -20167.072} C_VEL
LIN {X 0,Y 228.163,Z 378.059,A -85,B 0,C 180,E1 -20170.651,E2 -20170.651} C_VEL
LIN {X 0,Y 228.05,Z 378.076,A -85,B 0,C 180,E1 -20176.103,E2 -20176.103} C_VEL
LIN {X 0,Y 227.935,Z 378.089,A -85,B 0,C 180,E1 -20179.826,E2 -20179.826} C_VEL
LIN {X 0,Y 227.906,Z 378.096,A -85,B 0,C 180,E1 -20183.634,E2 -20183.634} C_VEL
LIN {X 0,Y 227.872,Z 378.098,A -85,B 0,C 180,E1 -20187.557,E2 -20187.557} C_VEL
LIN {X 0,Y 227.862,Z 378.101,A -85,B 0,C 180,E1 -20191.624,E2 -20191.624} C_VEL
LIN {X 0,Y 227.896,Z 378.094,A -85,B 0,C 180,E1 -20195.869,E2 -20195.869} C_VEL
LIN {X 0,Y 227.913,Z 378.093,A -85,B 0,C 180,E1 -20200.359,E2 -20200.359} C_VEL
LIN {X 0,Y 227.915,Z 378.093,A -85,B 0,C 180,E1 -20204.831,E2 -20204.831} C_VEL
LIN {X 0,Y 227.922,Z 378.092,A -85,B 0,C 180,E1 -20207.735,E2 -20207.735} C_VEL
LIN {X 0,Y 227.883,Z 378.097,A -85,B 0,C 180,E1 -20211.92,E2 -20211.92} C_VEL
LIN {X 0,Y 228.056,Z 378.136,A -85,B 0,C 180,E1 -20215.138,E2 -20215.138} C_VEL
LIN {X 0,Y 230.501,Z 390.664,A -85,B 0,C 180,E1 -20219.561,E2 -20219.561} C_VEL
LIN {X 0,Y 230.228,Z 393.238,A -85,B 0,C 180,E1 -20220.419,E2 -20220.419} C_VEL
LIN {X 0,Y 228.217,Z 396.627,A -85,B 0,C 180,E1 -20221.504,E2 -20221.504} C_VEL
LIN {X 0,Y 224.741,Z 401.494,A -85,B 0,C 180,E1 -20222.837,E2 -20222.837} C_VEL
LIN {X 0,Y 223.988,Z 404.185,A -85,B 0,C 180,E1 -20223.187,E2 -20223.187} C_VEL
LIN {X 0,Y 223.954,Z 404.787,A -85,B 0,C 180,E1 -20223.227,E2 -20223.227} C_VEL
LIN {X 0,Y 224.887,Z 427.311,A -85,B 0,C 180,E1 -20224.491,E2 -20224.491} C_VEL
LIN {X 0,Y 227.322,Z 457.588,A -85,B 0,C 180,E1 -20226.216,E2 -20226.216} C_VEL
LIN {X 0,Y 225.131,Z 511.693,A -85,B 0,C 180,E1 -20229.204,E2 -20229.204} C_VEL
LIN {X 0,Y 224.426,Z 524.203,A -85,B 0,C 180,E1 -20230.208,E2 -20230.208} C_VEL
LIN {X 0,Y 223.47,Z 536.258,A -85,B 0,C 180,E1 -20231.491,E2 -20231.491} C_VEL
LIN {X 0,Y 222.514,Z 549.021,A -85,B 0,C 180,E1 -20233.252,E2 -20233.252} C_VEL
LIN {X 0,Y 221.627,Z 559.588,A -85,B 0,C 180,E1 -20235.072,E2 -20235.072} C_VEL
LIN {X 0,Y 220.978,Z 569.341,A -85,B 0,C 180,E1 -20237.139,E2 -20237.139} C_VEL
LIN {X 0,Y 220.508,Z 578.288,A -85,B 0,C 180,E1 -20239.442,E2 -20239.442} C_VEL
LIN {X 0,Y 220.229,Z 586.313,A -85,B 0,C 180,E1 -20241.964,E2 -20241.964} C_VEL
LIN {X 0,Y 220.234,Z 592.868,A -85,B 0,C 180,E1 -20244.509,E2 -20244.509} C_VEL
LIN {X 0,Y 220.29,Z 598.415,A -85,B 0,C 180,E1 -20247.259,E2 -20247.259} C_VEL
LIN {X 0,Y 220.29,Z 602.6,A -85,B 0,C 180,E1 -20250.002,E2 -20250.002} C_VEL
LIN {X 0,Y 219.866,Z 604.606,A -85,B 0,C 180,E1 -20251.834,E2 -20251.834} C_VEL
LIN {X 0,Y 219.479,Z 606.164,A -85,B 0,C 180,E1 -20253.674,E2 -20253.674} C_VEL
LIN {X 0,Y 219.176,Z 607.619,A -85,B 0,C 180,E1 -20256.26,E2 -20256.26} C_VEL
LIN {X 0,Y 219.136,Z 608.333,A -85,B 0,C 180,E1 -20259.23,E2 -20259.23} C_VEL
LIN {X 0,Y 220.028,Z 607.877,A -85,B 0,C 180,E1 -20262.922,E2 -20262.922} C_VEL
LIN {X 0,Y 222.162,Z 605.987,A -85,B 0,C 180,E1 -20266.544,E2 -20266.544} C_VEL
LIN {X 0,Y 225.213,Z 602.604,A -85,B 0,C 180,E1 -20270.078,E2 -20270.078} C_VEL
LIN {X 0,Y 228.297,Z 599.08,A -85,B 0,C 180,E1 -20272.633,E2 -20272.633} C_VEL
LIN {X 0,Y 231.964,Z 594.615,A -85,B 0,C 180,E1 -20275.1,E2 -20275.1} C_VEL
LIN {X 0,Y 237.169,Z 588.138,A -85,B 0,C 180,E1 -20277.823,E2 -20277.823} C_VEL
LIN {X 0,Y 243.03,Z 580.11,A -85,B 0,C 180,E1 -20280.404,E2 -20280.404} C_VEL
LIN {X 0,Y 248.663,Z 571.81,A -85,B 0,C 180,E1 -20282.482,E2 -20282.482} C_VEL
LIN {X 0,Y 254.799,Z 561.943,A -85,B 0,C 180,E1 -20284.435,E2 -20284.435} C_VEL
LIN {X 0,Y 260.885,Z 551.257,A -85,B 0,C 180,E1 -20286.037,E2 -20286.037} C_VEL
LIN {X 0,Y 267.166,Z 538.896,A -85,B 0,C 180,E1 -20287.47,E2 -20287.47} C_VEL
LIN {X 0,Y 272.943,Z 525.605,A -85,B 0,C 180,E1 -20288.641,E2 -20288.641} C_VEL
LIN {X 0,Y 277.88,Z 511.995,A -85,B 0,C 180,E1 -20289.573,E2 -20289.573} C_VEL
LIN {X 0,Y 282.279,Z 496.765,A -85,B 0,C 180,E1 -20290.386,E2 -20290.386} C_VEL
LIN {X 0,Y 287.283,Z 474.67,A -85,B 0,C 180,E1 -20291.397,E2 -20291.397} C_VEL
LIN {X 0,Y 287.672,Z 472.14,A -85,B 0,C 180,E1 -20291.704,E2 -20291.704} C_VEL
LIN {X 0,Y 287.455,Z 467.458,A -85,B 0,C 180,E1 -20293.955,E2 -20293.955} C_VEL
LIN {X 0,Y 287.564,Z 465.52,A -85,B 0,C 180,E1 -20296.124,E2 -20296.124} C_VEL
LIN {X 0,Y 287.824,Z 465.07,A -85,B 0,C 180,E1 -20297.101,E2 -20297.101} C_VEL
LIN {X 0,Y 288.745,Z 465.456,A -85,B 0,C 180,E1 -20299.253,E2 -20299.253} C_VEL
LIN {X 0,Y 288.901,Z 465.654,A -85,B 0,C 180,E1 -20299.551,E2 -20299.551} C_VEL
LIN {X 0,Y 283.545,Z 488.723,A -85,B 0,C 180,E1 -20300.641,E2 -20300.641} C_VEL
LIN {X 0,Y 280.257,Z 500.648,A -85,B 0,C 180,E1 -20301.406,E2 -20301.406} C_VEL
LIN {X 0,Y 275.712,Z 513.78,A -85,B 0,C 180,E1 -20302.513,E2 -20302.513} C_VEL
LIN {X 0,Y 270.812,Z 525.494,A -85,B 0,C 180,E1 -20303.814,E2 -20303.814} C_VEL
LIN {X 0,Y 265.504,Z 536.308,A -85,B 0,C 180,E1 -20305.311,E2 -20305.311} C_VEL
LIN {X 0,Y 259.485,Z 546.863,A -85,B 0,C 180,E1 -20307.201,E2 -20307.201} C_VEL
LIN {X 0,Y 253.92,Z 555.358,A -85,B 0,C 180,E1 -20309.107,E2 -20309.107} C_VEL
LIN {X 0,Y 248.365,Z 562.777,A -85,B 0,C 180,E1 -20311.246,E2 -20311.246} C_VEL
LIN {X 0,Y 243.504,Z 568.588,A -85,B 0,C 180,E1 -20313.425,E2 -20313.425} C_VEL
LIN {X 0,Y 239.024,Z 573.283,A -85,B 0,C 180,E1 -20315.692,E2 -20315.692} C_VEL
LIN {X 0,Y 233.747,Z 577.98,A -85,B 0,C 180,E1 -20318.85,E2 -20318.85} C_VEL
LIN {X 0,Y 229.239,Z 580.956,A -85,B 0,C 180,E1 -20322.147,E2 -20322.147} C_VEL
LIN {X 0,Y 225.608,Z 582.383,A -85,B 0,C 180,E1 -20325.569,E2 -20325.569} C_VEL
LIN {X 0,Y 224.034,Z 582.514,A -85,B 0,C 180,E1 -20327.315,E2 -20327.315} C_VEL
LIN {X 0,Y 221.67,Z 581.561,A -85,B 0,C 180,E1 -20330.879,E2 -20330.879} C_VEL
LIN {X 0,Y 220.317,Z 579.069,A -85,B 0,C 180,E1 -20334.508,E2 -20334.508} C_VEL
LIN {X 0,Y 219.483,Z 576.108,A -85,B 0,C 180,E1 -20337.247,E2 -20337.247} C_VEL
LIN {X 0,Y 219.098,Z 572.144,A -85,B 0,C 180,E1 -20340,E2 -20340} C_VEL
LIN {X 0,Y 219.131,Z 567.091,A -85,B 0,C 180,E1 -20342.757,E2 -20342.757} C_VEL
LIN {X 0,Y 219.295,Z 561.906,A -85,B 0,C 180,E1 -20345.056,E2 -20345.056} C_VEL
LIN {X 0,Y 219.647,Z 554.387,A -85,B 0,C 180,E1 -20347.815,E2 -20347.815} C_VEL
LIN {X 0,Y 220.264,Z 545.049,A -85,B 0,C 180,E1 -20350.572,E2 -20350.572} C_VEL
LIN {X 0,Y 221.073,Z 534.583,A -85,B 0,C 180,E1 -20353.091,E2 -20353.091} C_VEL
LIN {X 0,Y 222.076,Z 522.779,A -85,B 0,C 180,E1 -20355.369,E2 -20355.369} C_VEL
LIN {X 0,Y 223.078,Z 511.186,A -85,B 0,C 180,E1 -20357.179,E2 -20357.179} C_VEL
LIN {X 0,Y 223.974,Z 497.337,A -85,B 0,C 180,E1 -20358.88,E2 -20358.88} C_VEL
LIN {X 0,Y 224.844,Z 483.425,A -85,B 0,C 180,E1 -20360.163,E2 -20360.163} C_VEL
LIN {X 0,Y 225.489,Z 468.664,A -85,B 0,C 180,E1 -20361.122,E2 -20361.122} C_VEL
LIN {X 0,Y 228.184,Z 404.73,A -85,B 0,C 180,E1 -20364.509,E2 -20364.509} C_VEL
LIN {X 0,Y 220.958,Z 378.984,A -85,B 0,C 180,E1 -20366.194,E2 -20366.194} C_VEL
LIN {X 0,Y 220.869,Z 378.97,A -85,B 0,C 180,E1 -20370.777,E2 -20370.777} C_VEL
LIN {X 0,Y 220.809,Z 378.978,A -85,B 0,C 180,E1 -20374.953,E2 -20374.953} C_VEL
LIN {X 0,Y 220.812,Z 378.977,A -85,B 0,C 180,E1 -20379.536,E2 -20379.536} C_VEL
LIN {X 0,Y 220.779,Z 378.984,A -85,B 0,C 180,E1 -20384.453,E2 -20384.453} C_VEL
LIN {X 0,Y 220.775,Z 378.985,A -85,B 0,C 180,E1 -20388.046,E2 -20388.046} C_VEL
LIN {X 0,Y 220.829,Z 378.976,A -85,B 0,C 180,E1 -20392.792,E2 -20392.792} C_VEL
LIN {X 0,Y 220.828,Z 378.975,A -85,B 0,C 180,E1 -20397.244,E2 -20397.244} C_VEL
LIN {X 0,Y 220.84,Z 378.973,A -85,B 0,C 180,E1 -20401.485,E2 -20401.485} C_VEL
LIN {X 0,Y 220.871,Z 378.971,A -85,B 0,C 180,E1 -20405.563,E2 -20405.563} C_VEL
LIN {X 0,Y 220.896,Z 378.966,A -85,B 0,C 180,E1 -20409.512,E2 -20409.512} C_VEL
LIN {X 0,Y 221.02,Z 378.952,A -85,B 0,C 180,E1 -20413.368,E2 -20413.368} C_VEL
LIN {X 0,Y 221.084,Z 378.943,A -85,B 0,C 180,E1 -20419.002,E2 -20419.002} C_VEL
LIN {X 0,Y 221.262,Z 378.922,A -85,B 0,C 180,E1 -20422.699,E2 -20422.699} C_VEL
LIN {X 0,Y 221.515,Z 378.893,A -85,B 0,C 180,E1 -20428.18,E2 -20428.18} C_VEL
LIN {X 0,Y 221.515,Z 378.893,A -85,B 0,C 180,E1 -20431.816,E2 -20431.816} C_VEL
LIN {X 0,Y 221.312,Z 378.915,A -85,B 0,C 180,E1 -20437.295,E2 -20437.295} C_VEL
LIN {X 0,Y 221.116,Z 378.939,A -85,B 0,C 180,E1 -20440.992,E2 -20440.992} C_VEL
LIN {X 0,Y 221.015,Z 378.953,A -85,B 0,C 180,E1 -20446.628,E2 -20446.628} C_VEL
LIN {X 0,Y 220.891,Z 378.966,A -85,B 0,C 180,E1 -20450.484,E2 -20450.484} C_VEL
LIN {X 0,Y 220.864,Z 378.972,A -85,B 0,C 180,E1 -20454.433,E2 -20454.433} C_VEL
LIN {X 0,Y 220.833,Z 378.974,A -85,B 0,C 180,E1 -20458.511,E2 -20458.511} C_VEL
LIN {X 0,Y 220.82,Z 378.976,A -85,B 0,C 180,E1 -20462.753,E2 -20462.753} C_VEL
LIN {X 0,Y 220.833,Z 378.976,A -85,B 0,C 180,E1 -20467.286,E2 -20467.286} C_VEL
LIN {X 0,Y 220.866,Z 378.974,A -85,B 0,C 180,E1 -20471.927,E2 -20471.927} C_VEL
LIN {X 0,Y 220.868,Z 378.973,A -85,B 0,C 180,E1 -20475.57,E2 -20475.57} C_VEL
LIN {X 0,Y 220.854,Z 378.974,A -85,B 0,C 180,E1 -20479.79,E2 -20479.79} C_VEL
LIN {X 0,Y 220.828,Z 378.976,A -85,B 0,C 180,E1 -20482.794,E2 -20482.794} C_VEL
LIN {X 0,Y 220.817,Z 378.975,A -85,B 0,C 180,E1 -20487.244,E2 -20487.244} C_VEL
LIN {X 0,Y 220.83,Z 378.978,A -85,B 0,C 180,E1 -20491.486,E2 -20491.486} C_VEL
LIN {X 0,Y 220.859,Z 378.972,A -85,B 0,C 180,E1 -20495.564,E2 -20495.564} C_VEL
LIN {X 0,Y 220.884,Z 378.972,A -85,B 0,C 180,E1 -20499.513,E2 -20499.513} C_VEL
LIN {X 0,Y 221.008,Z 378.955,A -85,B 0,C 180,E1 -20503.37,E2 -20503.37} C_VEL
LIN {X 0,Y 221.108,Z 378.942,A -85,B 0,C 180,E1 -20509.006,E2 -20509.006} C_VEL
LIN {X 0,Y 221.302,Z 378.914,A -85,B 0,C 180,E1 -20512.702,E2 -20512.702} C_VEL
LIN {X 0,Y 221.507,Z 378.892,A -85,B 0,C 180,E1 -20518.182,E2 -20518.182} C_VEL
LIN {X 0,Y 221.506,Z 378.89,A -85,B 0,C 180,E1 -20521.818,E2 -20521.818} C_VEL
LIN {X 0,Y 221.303,Z 378.919,A -85,B 0,C 180,E1 -20527.298,E2 -20527.298} C_VEL
LIN {X 0,Y 221.109,Z 378.939,A -85,B 0,C 180,E1 -20530.995,E2 -20530.995} C_VEL
LIN {X 0,Y 221.008,Z 378.953,A -85,B 0,C 180,E1 -20536.631,E2 -20536.631} C_VEL
LIN {X 0,Y 220.885,Z 378.966,A -85,B 0,C 180,E1 -20540.487,E2 -20540.487} C_VEL
LIN {X 0,Y 220.86,Z 378.972,A -85,B 0,C 180,E1 -20544.436,E2 -20544.436} C_VEL
LIN {X 0,Y 220.82,Z 378.973,A -85,B 0,C 180,E1 -20548.516,E2 -20548.516} C_VEL
LIN {X 0,Y 220.816,Z 378.978,A -85,B 0,C 180,E1 -20552.757,E2 -20552.757} C_VEL
LIN {X 0,Y 220.862,Z 378.971,A -85,B 0,C 180,E1 -20557.3,E2 -20557.3} C_VEL
LIN {X 0,Y 220.873,Z 378.971,A -85,B 0,C 180,E1 -20561.929,E2 -20561.929} C_VEL
LIN {X 0,Y 220.869,Z 378.969,A -85,B 0,C 180,E1 -20565.574,E2 -20565.574} C_VEL
LIN {X 0,Y 220.854,Z 378.973,A -85,B 0,C 180,E1 -20569.794,E2 -20569.794} C_VEL
LIN {X 0,Y 221.025,Z 379.117,A -85,B 0,C 180,E1 -20575.088,E2 -20575.088} C_VEL
LIN {X 0,Y 224.093,Z 394.409,A -85,B 0,C 180,E1 -20580.62,E2 -20580.62} C_VEL
LIN {X 0,Y 224.654,Z 397.321,A -85,B 0,C 180,E1 -20581.641,E2 -20581.641} C_VEL
LIN {X 0,Y 224.049,Z 401.363,A -85,B 0,C 180,E1 -20583.011,E2 -20583.011} C_VEL
LIN {X 0,Y 223.954,Z 404.787,A -85,B 0,C 180,E1 -20583.227,E2 -20583.227} C_VEL
LIN {X 0,Y 223.294,Z 410.564,A -85,B 0,C 180,E1 -20583.518,E2 -20583.518} C_VEL
LIN {X 0,Y 218.532,Z 429.453,A -85,B 0,C 180,E1 -20584.418,E2 -20584.418} C_VEL
LIN {X 0,Y 218.332,Z 435.192,A -85,B 0,C 180,E1 -20584.742,E2 -20584.742} C_VEL
LIN {X 0,Y 220.258,Z 457.444,A -85,B 0,C 180,E1 -20586.059,E2 -20586.059} C_VEL
LIN {X 0,Y 218.049,Z 511.488,A -85,B 0,C 180,E1 -20589.182,E2 -20589.182} C_VEL
LIN {X 0,Y 217.343,Z 523.755,A -85,B 0,C 180,E1 -20590.214,E2 -20590.214} C_VEL
LIN {X 0,Y 216.408,Z 535.741,A -85,B 0,C 180,E1 -20591.543,E2 -20591.543} C_VEL
LIN {X 0,Y 215.423,Z 548.767,A -85,B 0,C 180,E1 -20593.416,E2 -20593.416} C_VEL
LIN {X 0,Y 214.58,Z 559.234,A -85,B 0,C 180,E1 -20595.298,E2 -20595.298} C_VEL
LIN {X 0,Y 213.864,Z 569.89,A -85,B 0,C 180,E1 -20597.669,E2 -20597.669} C_VEL
LIN {X 0,Y 213.471,Z 578.62,A -85,B 0,C 180,E1 -20600.049,E2 -20600.049} C_VEL
LIN {X 0,Y 213.3,Z 587.081,A -85,B 0,C 180,E1 -20602.905,E2 -20602.905} C_VEL
LIN {X 0,Y 213.34,Z 592.78,A -85,B 0,C 180,E1 -20605.278,E2 -20605.278} C_VEL
LIN {X 0,Y 213.377,Z 598.143,A -85,B 0,C 180,E1 -20608.115,E2 -20608.115} C_VEL
LIN {X 0,Y 213.354,Z 600.962,A -85,B 0,C 180,E1 -20610.002,E2 -20610.002} C_VEL
LIN {X 0,Y 212.916,Z 603.158,A -85,B 0,C 180,E1 -20611.894,E2 -20611.894} C_VEL
LIN {X 0,Y 212.494,Z 604.833,A -85,B 0,C 180,E1 -20613.795,E2 -20613.795} C_VEL
LIN {X 0,Y 212.169,Z 606.473,A -85,B 0,C 180,E1 -20616.414,E2 -20616.414} C_VEL
LIN {X 0,Y 212.138,Z 607.434,A -85,B 0,C 180,E1 -20619.537,E2 -20619.537} C_VEL
LIN {X 0,Y 213.086,Z 607.324,A -85,B 0,C 180,E1 -20623.351,E2 -20623.351} C_VEL
LIN {X 0,Y 215.328,Z 605.752,A -85,B 0,C 180,E1 -20627.085,E2 -20627.085} C_VEL
LIN {X 0,Y 218.546,Z 602.754,A -85,B 0,C 180,E1 -20630.718,E2 -20630.718} C_VEL
LIN {X 0,Y 221.795,Z 599.544,A -85,B 0,C 180,E1 -20633.336,E2 -20633.336} C_VEL
LIN {X 0,Y 225.622,Z 595.468,A -85,B 0,C 180,E1 -20635.857,E2 -20635.857} C_VEL
LIN {X 0,Y 231.834,Z 588.488,A -85,B 0,C 180,E1 -20639.017,E2 -20639.017} C_VEL
LIN {X 0,Y 238.026,Z 580.859,A -85,B 0,C 180,E1 -20641.609,E2 -20641.609} C_VEL
LIN {X 0,Y 243.946,Z 572.921,A -85,B 0,C 180,E1 -20643.684,E2 -20643.684} C_VEL
LIN {X 0,Y 251.49,Z 561.747,A -85,B 0,C 180,E1 -20645.936,E2 -20645.936} C_VEL
LIN {X 0,Y 257.598,Z 551.82,A -85,B 0,C 180,E1 -20647.437,E2 -20647.437} C_VEL
LIN {X 0,Y 264.401,Z 539.282,A -85,B 0,C 180,E1 -20648.902,E2 -20648.902} C_VEL
LIN {X 0,Y 270.428,Z 526.454,A -85,B 0,C 180,E1 -20650.034,E2 -20650.034} C_VEL
LIN {X 0,Y 276.254,Z 511.501,A -85,B 0,C 180,E1 -20651.049,E2 -20651.049} C_VEL
LIN {X 0,Y 280.776,Z 496.848,A -85,B 0,C 180,E1 -20651.808,E2 -20651.808} C_VEL
LIN {X 0,Y 285.509,Z 477.262,A -85,B 0,C 180,E1 -20652.682,E2 -20652.682} C_VEL
LIN {X 0,Y 285.541,Z 474.096,A -85,B 0,C 180,E1 -20654.298,E2 -20654.298} C_VEL
LIN {X 0,Y 285.778,Z 472.246,A -85,B 0,C 180,E1 -20656.481,E2 -20656.481} C_VEL
LIN {X 0,Y 286.357,Z 472.004,A -85,B 0,C 180,E1 -20658.199,E2 -20658.199} C_VEL
LIN {X 0,Y 286.447,Z 472.023,A -85,B 0,C 180,E1 -20658.402,E2 -20658.402} C_VEL
LIN {X 0,Y 281.572,Z 491.754,A -85,B 0,C 180,E1 -20659.356,E2 -20659.356} C_VEL
LIN {X 0,Y 277.289,Z 505.515,A -85,B 0,C 180,E1 -20660.287,E2 -20660.287} C_VEL
LIN {X 0,Y 272.157,Z 518.568,A -85,B 0,C 180,E1 -20661.465,E2 -20661.465} C_VEL
LIN {X 0,Y 267.017,Z 529.54,A -85,B 0,C 180,E1 -20662.744,E2 -20662.744} C_VEL
LIN {X 0,Y 261.49,Z 539.641,A -85,B 0,C 180,E1 -20664.227,E2 -20664.227} C_VEL
LIN {X 0,Y 255.192,Z 549.699,A -85,B 0,C 180,E1 -20666.104,E2 -20666.104} C_VEL
LIN {X 0,Y 249.159,Z 557.99,A -85,B 0,C 180,E1 -20668.07,E2 -20668.07} C_VEL
LIN {X 0,Y 242.643,Z 565.86,A -85,B 0,C 180,E1 -20670.502,E2 -20670.502} C_VEL
LIN {X 0,Y 235.924,Z 572.754,A -85,B 0,C 180,E1 -20673.459,E2 -20673.459} C_VEL
LIN {X 0,Y 231.621,Z 576.522,A -85,B 0,C 180,E1 -20675.678,E2 -20675.678} C_VEL
LIN {X 0,Y 227.326,Z 579.68,A -85,B 0,C 180,E1 -20678.223,E2 -20678.223} C_VEL
LIN {X 0,Y 222.627,Z 582.27,A -85,B 0,C 180,E1 -20681.598,E2 -20681.598} C_VEL
LIN {X 0,Y 218.792,Z 583.262,A -85,B 0,C 180,E1 -20685.109,E2 -20685.109} C_VEL
LIN {X 0,Y 215.772,Z 582.761,A -85,B 0,C 180,E1 -20688.73,E2 -20688.73} C_VEL
LIN {X 0,Y 214.692,Z 581.921,A -85,B 0,C 180,E1 -20690.579,E2 -20690.579} C_VEL
LIN {X 0,Y 213.263,Z 579.033,A -85,B 0,C 180,E1 -20694.326,E2 -20694.326} C_VEL
LIN {X 0,Y 212.408,Z 575.805,A -85,B 0,C 180,E1 -20697.155,E2 -20697.155} C_VEL
LIN {X 0,Y 212.02,Z 571.57,A -85,B 0,C 180,E1 -20700,E2 -20700} C_VEL
LIN {X 0,Y 212.119,Z 565.214,A -85,B 0,C 180,E1 -20703.324,E2 -20703.324} C_VEL
LIN {X 0,Y 212.25,Z 559.56,A -85,B 0,C 180,E1 -20705.701,E2 -20705.701} C_VEL
LIN {X 0,Y 212.731,Z 551.377,A -85,B 0,C 180,E1 -20708.549,E2 -20708.549} C_VEL
LIN {X 0,Y 213.436,Z 541.234,A -85,B 0,C 180,E1 -20711.395,E2 -20711.395} C_VEL
LIN {X 0,Y 214.277,Z 530.901,A -85,B 0,C 180,E1 -20713.756,E2 -20713.756} C_VEL
LIN {X 0,Y 215.253,Z 519.505,A -85,B 0,C 180,E1 -20715.869,E2 -20715.869} C_VEL
LIN {X 0,Y 216.244,Z 507.041,A -85,B 0,C 180,E1 -20717.739,E2 -20717.739} C_VEL
LIN {X 0,Y 217.161,Z 493.166,A -85,B 0,C 180,E1 -20719.348,E2 -20719.348} C_VEL
LIN {X 0,Y 218.026,Z 478.705,A -85,B 0,C 180,E1 -20720.581,E2 -20720.581} C_VEL
LIN {X 0,Y 219.77,Z 435.524,A -85,B 0,C 180,E1 -20723.063,E2 -20723.063} C_VEL
LIN {X 0,Y 221.145,Z 406,A -85,B 0,C 180,E1 -20724.684,E2 -20724.684} C_VEL
LIN {X 0,Y 213.874,Z 379.845,A -85,B 0,C 180,E1 -20726.47,E2 -20726.47} C_VEL
LIN {X 0,Y 213.784,Z 379.852,A -85,B 0,C 180,E1 -20731.735,E2 -20731.735} C_VEL
LIN {X 0,Y 213.75,Z 379.861,A -85,B 0,C 180,E1 -20736.287,E2 -20736.287} C_VEL
LIN {X 0,Y 213.717,Z 379.858,A -85,B 0,C 180,E1 -20741.124,E2 -20741.124} C_VEL
LIN {X 0,Y 213.711,Z 379.861,A -85,B 0,C 180,E1 -20743.677,E2 -20743.677} C_VEL
LIN {X 0,Y 213.711,Z 379.865,A -85,B 0,C 180,E1 -20746.343,E2 -20746.343} C_VEL
LIN {X 0,Y 213.739,Z 379.856,A -85,B 0,C 180,E1 -20751.334,E2 -20751.334} C_VEL
LIN {X 0,Y 213.773,Z 379.857,A -85,B 0,C 180,E1 -20756.018,E2 -20756.018} C_VEL
LIN {X 0,Y 213.785,Z 379.854,A -85,B 0,C 180,E1 -20760.452,E2 -20760.452} C_VEL
LIN {X 0,Y 213.805,Z 379.851,A -85,B 0,C 180,E1 -20764.7,E2 -20764.7} C_VEL
LIN {X 0,Y 213.817,Z 379.847,A -85,B 0,C 180,E1 -20768.802,E2 -20768.802} C_VEL
LIN {X 0,Y 213.947,Z 379.833,A -85,B 0,C 180,E1 -20772.802,E2 -20772.802} C_VEL
LIN {X 0,Y 213.956,Z 379.829,A -85,B 0,C 180,E1 -20776.705,E2 -20776.705} C_VEL
LIN {X 0,Y 214.144,Z 379.809,A -85,B 0,C 180,E1 -20780.553,E2 -20780.553} C_VEL
LIN {X 0,Y 214.104,Z 379.812,A -85,B 0,C 180,E1 -20784.346,E2 -20784.346} C_VEL
LIN {X 0,Y 214.448,Z 379.773,A -85,B 0,C 180,E1 -20788.12,E2 -20788.12} C_VEL
LIN {X 0,Y 214.556,Z 379.761,A -85,B 0,C 180,E1 -20789.998,E2 -20789.998} C_VEL
LIN {X 0,Y 214.448,Z 379.773,A -85,B 0,C 180,E1 -20791.876,E2 -20791.876} C_VEL
LIN {X 0,Y 214.249,Z 379.796,A -85,B 0,C 180,E1 -20797.537,E2 -20797.537} C_VEL
LIN {X 0,Y 214.047,Z 379.82,A -85,B 0,C 180,E1 -20801.359,E2 -20801.359} C_VEL
LIN {X 0,Y 213.933,Z 379.834,A -85,B 0,C 180,E1 -20805.235,E2 -20805.235} C_VEL
LIN {X 0,Y 213.838,Z 379.846,A -85,B 0,C 180,E1 -20809.185,E2 -20809.185} C_VEL
LIN {X 0,Y 213.845,Z 379.844,A -85,B 0,C 180,E1 -20813.225,E2 -20813.225} C_VEL
LIN {X 0,Y 213.826,Z 379.849,A -85,B 0,C 180,E1 -20817.448,E2 -20817.448} C_VEL
LIN {X 0,Y 213.775,Z 379.854,A -85,B 0,C 180,E1 -20821.733,E2 -20821.733} C_VEL
LIN {X 0,Y 213.75,Z 379.858,A -85,B 0,C 180,E1 -20826.284,E2 -20826.284} C_VEL
LIN {X 0,Y 213.818,Z 379.847,A -85,B 0,C 180,E1 -20831.097,E2 -20831.097} C_VEL
LIN {X 0,Y 213.83,Z 379.851,A -85,B 0,C 180,E1 -20833.691,E2 -20833.691} C_VEL
LIN {X 0,Y 213.834,Z 379.846,A -85,B 0,C 180,E1 -20836.354,E2 -20836.354} C_VEL
LIN {X 0,Y 213.817,Z 379.846,A -85,B 0,C 180,E1 -20839.108,E2 -20839.108} C_VEL
LIN {X 0,Y 213.747,Z 379.861,A -85,B 0,C 180,E1 -20843.713,E2 -20843.713} C_VEL
LIN {X 0,Y 213.788,Z 379.851,A -85,B 0,C 180,E1 -20848.723,E2 -20848.723} C_VEL
LIN {X 0,Y 213.818,Z 379.849,A -85,B 0,C 180,E1 -20852.602,E2 -20852.602} C_VEL
LIN {X 0,Y 213.844,Z 379.843,A -85,B 0,C 180,E1 -20856.952,E2 -20856.952} C_VEL
LIN {X 0,Y 213.935,Z 379.833,A -85,B 0,C 180,E1 -20862.803,E2 -20862.803} C_VEL
LIN {X 0,Y 213.972,Z 379.829,A -85,B 0,C 180,E1 -20866.708,E2 -20866.708} C_VEL
LIN {X 0,Y 214.187,Z 379.802,A -85,B 0,C 180,E1 -20870.557,E2 -20870.557} C_VEL
LIN {X 0,Y 214.239,Z 379.794,A -85,B 0,C 180,E1 -20872.46,E2 -20872.46} C_VEL
LIN {X 0,Y 214.44,Z 379.772,A -85,B 0,C 180,E1 -20878.122,E2 -20878.122} C_VEL
LIN {X 0,Y 214.546,Z 379.758,A -85,B 0,C 180,E1 -20880,E2 -20880} C_VEL
LIN {X 0,Y 214.439,Z 379.77,A -85,B 0,C 180,E1 -20881.878,E2 -20881.878} C_VEL
LIN {X 0,Y 214.24,Z 379.799,A -85,B 0,C 180,E1 -20887.54,E2 -20887.54} C_VEL
LIN {X 0,Y 214.039,Z 379.821,A -85,B 0,C 180,E1 -20891.362,E2 -20891.362} C_VEL
LIN {X 0,Y 213.926,Z 379.838,A -85,B 0,C 180,E1 -20895.238,E2 -20895.238} C_VEL
LIN {X 0,Y 213.86,Z 379.844,A -85,B 0,C 180,E1 -20899.186,E2 -20899.186} C_VEL
LIN {X 0,Y 213.84,Z 379.849,A -85,B 0,C 180,E1 -20903.228,E2 -20903.228} C_VEL
LIN {X 0,Y 213.822,Z 379.848,A -85,B 0,C 180,E1 -20907.451,E2 -20907.451} C_VEL
LIN {X 0,Y 213.763,Z 379.857,A -85,B 0,C 180,E1 -20911.739,E2 -20911.739} C_VEL
LIN {X 0,Y 213.754,Z 379.854,A -85,B 0,C 180,E1 -20916.287,E2 -20916.287} C_VEL
LIN {X 0,Y 213.824,Z 379.851,A -85,B 0,C 180,E1 -20921.099,E2 -20921.099} C_VEL
LIN {X 0,Y 213.831,Z 379.847,A -85,B 0,C 180,E1 -20923.695,E2 -20923.695} C_VEL
LIN {X 0,Y 213.836,Z 379.843,A -85,B 0,C 180,E1 -20926.358,E2 -20926.358} C_VEL
LIN {X 0,Y 213.817,Z 379.851,A -85,B 0,C 180,E1 -20929.112,E2 -20929.112} C_VEL
LIN {X 0,Y 213.984,Z 379.959,A -85,B 0,C 180,E1 -20934.999,E2 -20934.999} C_VEL
LIN {X 0,Y 217.225,Z 395.942,A -85,B 0,C 180,E1 -20940.97,E2 -20940.97} C_VEL
LIN {X 0,Y 217.54,Z 397.535,A -85,B 0,C 180,E1 -20941.544,E2 -20941.544} C_VEL
LIN {X 0,Y 217.063,Z 400.899,A -85,B 0,C 180,E1 -20942.722,E2 -20942.722} C_VEL
LIN {X 0,Y 217.246,Z 417.583,A -85,B 0,C 180,E1 -20943.701,E2 -20943.701} C_VEL
LIN {X 0,Y 218.332,Z 435.192,A -85,B 0,C 180,E1 -20944.742,E2 -20944.742} C_VEL
LIN {X 0,Y 218.164,Z 440.976,A -85,B 0,C 180,E1 -20945.07,E2 -20945.07} C_VEL
LIN {X 0,Y 216.065,Z 450.494,A -85,B 0,C 180,E1 -20945.57,E2 -20945.57} C_VEL
LIN {X 0,Y 213.246,Z 461.942,A -85,B 0,C 180,E1 -20946.19,E2 -20946.19} C_VEL
LIN {X 0,Y 212.831,Z 465.826,A -85,B 0,C 180,E1 -20946.415,E2 -20946.415} C_VEL
LIN {X 0,Y 210.971,Z 511.528,A -85,B 0,C 180,E1 -20949.208,E2 -20949.208} C_VEL
LIN {X 0,Y 210.252,Z 523.642,A -85,B 0,C 180,E1 -20950.278,E2 -20950.278} C_VEL
LIN {X 0,Y 209.307,Z 535.477,A -85,B 0,C 180,E1 -20951.654,E2 -20951.654} C_VEL
LIN {X 0,Y 208.342,Z 548.378,A -85,B 0,C 180,E1 -20953.592,E2 -20953.592} C_VEL
LIN {X 0,Y 207.535,Z 558.762,A -85,B 0,C 180,E1 -20955.54,E2 -20955.54} C_VEL
LIN {X 0,Y 206.93,Z 568.398,A -85,B 0,C 180,E1 -20957.747,E2 -20957.747} C_VEL
LIN {X 0,Y 206.54,Z 577.255,A -85,B 0,C 180,E1 -20960.207,E2 -20960.207} C_VEL
LIN {X 0,Y 206.382,Z 585.844,A -85,B 0,C 180,E1 -20963.157,E2 -20963.157} C_VEL
LIN {X 0,Y 206.442,Z 592.597,A -85,B 0,C 180,E1 -20966.098,E2 -20966.098} C_VEL
LIN {X 0,Y 206.475,Z 597.796,A -85,B 0,C 180,E1 -20969.027,E2 -20969.027} C_VEL
LIN {X 0,Y 206.24,Z 600.468,A -85,B 0,C 180,E1 -20970.979,E2 -20970.979} C_VEL
LIN {X 0,Y 205.536,Z 603.393,A -85,B 0,C 180,E1 -20973.924,E2 -20973.924} C_VEL
LIN {X 0,Y 205.179,Z 605.225,A -85,B 0,C 180,E1 -20976.614,E2 -20976.614} C_VEL
LIN {X 0,Y 205.154,Z 606.458,A -85,B 0,C 180,E1 -20979.865,E2 -20979.865} C_VEL
LIN {X 0,Y 206.17,Z 606.64,A -85,B 0,C 180,E1 -20983.807,E2 -20983.807} C_VEL
LIN {X 0,Y 208.519,Z 605.444,A -85,B 0,C 180,E1 -20987.661,E2 -20987.661} C_VEL
LIN {X 0,Y 211.895,Z 602.862,A -85,B 0,C 180,E1 -20991.4,E2 -20991.4} C_VEL
LIN {X 0,Y 215.32,Z 599.957,A -85,B 0,C 180,E1 -20994.081,E2 -20994.081} C_VEL
LIN {X 0,Y 219.293,Z 596.229,A -85,B 0,C 180,E1 -20996.661,E2 -20996.661} C_VEL
LIN {X 0,Y 225.754,Z 589.838,A -85,B 0,C 180,E1 -20999.876,E2 -20999.876} C_VEL
LIN {X 0,Y 232.17,Z 582.764,A -85,B 0,C 180,E1 -21002.503,E2 -21002.503} C_VEL
LIN {X 0,Y 239.342,Z 574.069,A -85,B 0,C 180,E1 -21004.933,E2 -21004.933} C_VEL
LIN {X 0,Y 246.986,Z 563.778,A -85,B 0,C 180,E1 -21007.124,E2 -21007.124} C_VEL
LIN {X 0,Y 253.693,Z 553.799,A -85,B 0,C 180,E1 -21008.702,E2 -21008.702} C_VEL
LIN {X 0,Y 260.555,Z 542.376,A -85,B 0,C 180,E1 -21010.092,E2 -21010.092} C_VEL
LIN {X 0,Y 266.747,Z 530.517,A -85,B 0,C 180,E1 -21011.201,E2 -21011.201} C_VEL
LIN {X 0,Y 273.098,Z 516.112,A -85,B 0,C 180,E1 -21012.247,E2 -21012.247} C_VEL
LIN {X 0,Y 278.635,Z 500.463,A -85,B 0,C 180,E1 -21013.095,E2 -21013.095} C_VEL
LIN {X 0,Y 283.534,Z 482.024,A -85,B 0,C 180,E1 -21013.953,E2 -21013.953} C_VEL
LIN {X 0,Y 283.642,Z 480.561,A -85,B 0,C 180,E1 -21014.826,E2 -21014.826} C_VEL
LIN {X 0,Y 284.038,Z 478.954,A -85,B 0,C 180,E1 -21016.883,E2 -21016.883} C_VEL
LIN {X 0,Y 284.165,Z 478.811,A -85,B 0,C 180,E1 -21017.245,E2 -21017.245} C_VEL
LIN {X 0,Y 279.608,Z 495.767,A -85,B 0,C 180,E1 -21018.113,E2 -21018.113} C_VEL
LIN {X 0,Y 274.867,Z 509.319,A -85,B 0,C 180,E1 -21019.065,E2 -21019.065} C_VEL
LIN {X 0,Y 269.93,Z 520.828,A -85,B 0,C 180,E1 -21020.122,E2 -21020.122} C_VEL
LIN {X 0,Y 263.951,Z 532.486,A -85,B 0,C 180,E1 -21021.509,E2 -21021.509} C_VEL
LIN {X 0,Y 257.6,Z 543.086,A -85,B 0,C 180,E1 -21023.114,E2 -21023.114} C_VEL
LIN {X 0,Y 251.171,Z 552.338,A -85,B 0,C 180,E1 -21024.919,E2 -21024.919} C_VEL
LIN {X 0,Y 244.705,Z 560.474,A -85,B 0,C 180,E1 -21026.928,E2 -21026.928} C_VEL
LIN {X 0,Y 238.782,Z 566.968,A -85,B 0,C 180,E1 -21028.997,E2 -21028.997} C_VEL
LIN {X 0,Y 233.351,Z 572.223,A -85,B 0,C 180,E1 -21031.191,E2 -21031.191} C_VEL
LIN {X 0,Y 228.307,Z 576.447,A -85,B 0,C 180,E1 -21033.49,E2 -21033.49} C_VEL
LIN {X 0,Y 223.783,Z 579.684,A -85,B 0,C 180,E1 -21035.903,E2 -21035.903} C_VEL
LIN {X 0,Y 220.942,Z 581.34,A -85,B 0,C 180,E1 -21037.56,E2 -21037.56} C_VEL
LIN {X 0,Y 216.014,Z 583.464,A -85,B 0,C 180,E1 -21041.013,E2 -21041.013} C_VEL
LIN {X 0,Y 211.987,Z 584.099,A -85,B 0,C 180,E1 -21044.62,E2 -21044.62} C_VEL
LIN {X 0,Y 208.831,Z 583.172,A -85,B 0,C 180,E1 -21048.35,E2 -21048.35} C_VEL
LIN {X 0,Y 206.883,Z 580.736,A -85,B 0,C 180,E1 -21052.19,E2 -21052.19} C_VEL
LIN {X 0,Y 205.875,Z 577.858,A -85,B 0,C 180,E1 -21055.104,E2 -21055.104} C_VEL
LIN {X 0,Y 205.143,Z 574.017,A -85,B 0,C 180,E1 -21058.036,E2 -21058.036} C_VEL
LIN {X 0,Y 204.912,Z 569.119,A -85,B 0,C 180,E1 -21060.982,E2 -21060.982} C_VEL
LIN {X 0,Y 205.13,Z 563.061,A -85,B 0,C 180,E1 -21063.929,E2 -21063.929} C_VEL
LIN {X 0,Y 205.444,Z 554.571,A -85,B 0,C 180,E1 -21067.212,E2 -21067.212} C_VEL
LIN {X 0,Y 205.947,Z 546.278,A -85,B 0,C 180,E1 -21069.824,E2 -21069.824} C_VEL
LIN {X 0,Y 206.744,Z 535.879,A -85,B 0,C 180,E1 -21072.516,E2 -21072.516} C_VEL
LIN {X 0,Y 207.739,Z 524.214,A -85,B 0,C 180,E1 -21074.949,E2 -21074.949} C_VEL
LIN {X 0,Y 208.67,Z 512.806,A -85,B 0,C 180,E1 -21076.887,E2 -21076.887} C_VEL
LIN {X 0,Y 209.565,Z 500.236,A -85,B 0,C 180,E1 -21078.578,E2 -21078.578} C_VEL
LIN {X 0,Y 210.415,Z 487.166,A -85,B 0,C 180,E1 -21079.95,E2 -21079.95} C_VEL
LIN {X 0,Y 211.123,Z 473.368,A -85,B 0,C 180,E1 -21081,E2 -21081} C_VEL
LIN {X 0,Y 214.052,Z 406.938,A -85,B 0,C 180,E1 -21084.863,E2 -21084.863} C_VEL
LIN {X 0,Y 206.813,Z 380.723,A -85,B 0,C 180,E1 -21086.714,E2 -21086.714} C_VEL
LIN {X 0,Y 206.733,Z 380.731,A -85,B 0,C 180,E1 -21091.797,E2 -21091.797} C_VEL
LIN {X 0,Y 206.705,Z 380.734,A -85,B 0,C 180,E1 -21095.31,E2 -21095.31} C_VEL
LIN {X 0,Y 206.666,Z 380.74,A -85,B 0,C 180,E1 -21100.25,E2 -21100.25} C_VEL
LIN {X 0,Y 206.638,Z 380.746,A -85,B 0,C 180,E1 -21104.417,E2 -21104.417} C_VEL
LIN {X 0,Y 206.668,Z 380.738,A -85,B 0,C 180,E1 -21109.748,E2 -21109.748} C_VEL
LIN {X 0,Y 206.736,Z 380.732,A -85,B 0,C 180,E1 -21114.693,E2 -21114.693} C_VEL
LIN {X 0,Y 206.728,Z 380.728,A -85,B 0,C 180,E1 -21119.337,E2 -21119.337} C_VEL
LIN {X 0,Y 206.737,Z 380.733,A -85,B 0,C 180,E1 -21123.77,E2 -21123.77} C_VEL
LIN {X 0,Y 206.762,Z 380.727,A -85,B 0,C 180,E1 -21128.041,E2 -21128.041} C_VEL
LIN {X 0,Y 206.877,Z 380.717,A -85,B 0,C 180,E1 -21132.195,E2 -21132.195} C_VEL
LIN {X 0,Y 206.899,Z 380.709,A -85,B 0,C 180,E1 -21136.242,E2 -21136.242} C_VEL
LIN {X 0,Y 207.101,Z 380.688,A -85,B 0,C 180,E1 -21140.229,E2 -21140.229} C_VEL
LIN {X 0,Y 207.065,Z 380.69,A -85,B 0,C 180,E1 -21144.154,E2 -21144.154} C_VEL
LIN {X 0,Y 207.385,Z 380.653,A -85,B 0,C 180,E1 -21148.056,E2 -21148.056} C_VEL
LIN {X 0,Y 207.521,Z 380.637,A -85,B 0,C 180,E1 -21149.998,E2 -21149.998} C_VEL
LIN {X 0,Y 207.089,Z 380.687,A -85,B 0,C 180,E1 -21153.89,E2 -21153.89} C_VEL
LIN {X 0,Y 207.189,Z 380.677,A -85,B 0,C 180,E1 -21157.796,E2 -21157.796} C_VEL
LIN {X 0,Y 206.983,Z 380.702,A -85,B 0,C 180,E1 -21161.753,E2 -21161.753} C_VEL
LIN {X 0,Y 206.866,Z 380.716,A -85,B 0,C 180,E1 -21165.768,E2 -21165.768} C_VEL
LIN {X 0,Y 206.782,Z 380.727,A -85,B 0,C 180,E1 -21169.867,E2 -21169.867} C_VEL
LIN {X 0,Y 206.761,Z 380.73,A -85,B 0,C 180,E1 -21174.07,E2 -21174.07} C_VEL
LIN {X 0,Y 206.74,Z 380.73,A -85,B 0,C 180,E1 -21178.416,E2 -21178.416} C_VEL
LIN {X 0,Y 206.705,Z 380.734,A -85,B 0,C 180,E1 -21182.953,E2 -21182.953} C_VEL
LIN {X 0,Y 206.721,Z 380.734,A -85,B 0,C 180,E1 -21187.728,E2 -21187.728} C_VEL
LIN {X 0,Y 206.743,Z 380.731,A -85,B 0,C 180,E1 -21191.594,E2 -21191.594} C_VEL
LIN {X 0,Y 206.74,Z 380.733,A -85,B 0,C 180,E1 -21195.548,E2 -21195.548} C_VEL
LIN {X 0,Y 206.737,Z 380.732,A -85,B 0,C 180,E1 -21199.767,E2 -21199.767} C_VEL
LIN {X 0,Y 206.724,Z 380.732,A -85,B 0,C 180,E1 -21204.694,E2 -21204.694} C_VEL
LIN {X 0,Y 206.716,Z 380.734,A -85,B 0,C 180,E1 -21209.338,E2 -21209.338} C_VEL
LIN {X 0,Y 206.725,Z 380.733,A -85,B 0,C 180,E1 -21213.771,E2 -21213.771} C_VEL
LIN {X 0,Y 206.75,Z 380.73,A -85,B 0,C 180,E1 -21218.043,E2 -21218.043} C_VEL
LIN {X 0,Y 206.865,Z 380.715,A -85,B 0,C 180,E1 -21222.196,E2 -21222.196} C_VEL
LIN {X 0,Y 206.905,Z 380.709,A -85,B 0,C 180,E1 -21226.245,E2 -21226.245} C_VEL
LIN {X 0,Y 207.124,Z 380.683,A -85,B 0,C 180,E1 -21230.232,E2 -21230.232} C_VEL
LIN {X 0,Y 207.18,Z 380.673,A -85,B 0,C 180,E1 -21232.202,E2 -21232.202} C_VEL
LIN {X 0,Y 207.377,Z 380.652,A -85,B 0,C 180,E1 -21238.058,E2 -21238.058} C_VEL
LIN {X 0,Y 207.511,Z 380.634,A -85,B 0,C 180,E1 -21240,E2 -21240} C_VEL
LIN {X 0,Y 207.081,Z 380.689,A -85,B 0,C 180,E1 -21243.892,E2 -21243.892} C_VEL
LIN {X 0,Y 207.181,Z 380.677,A -85,B 0,C 180,E1 -21247.799,E2 -21247.799} C_VEL
LIN {X 0,Y 206.975,Z 380.701,A -85,B 0,C 180,E1 -21251.756,E2 -21251.756} C_VEL
LIN {X 0,Y 206.859,Z 380.717,A -85,B 0,C 180,E1 -21255.772,E2 -21255.772} C_VEL
LIN {X 0,Y 206.792,Z 380.722,A -85,B 0,C 180,E1 -21259.869,E2 -21259.869} C_VEL
LIN {X 0,Y 206.756,Z 380.729,A -85,B 0,C 180,E1 -21264.073,E2 -21264.073} C_VEL
LIN {X 0,Y 206.73,Z 380.728,A -85,B 0,C 180,E1 -21268.421,E2 -21268.421} C_VEL
LIN {X 0,Y 206.699,Z 380.737,A -85,B 0,C 180,E1 -21272.958,E2 -21272.958} C_VEL
LIN {X 0,Y 206.74,Z 380.729,A -85,B 0,C 180,E1 -21277.727,E2 -21277.727} C_VEL
LIN {X 0,Y 206.748,Z 380.731,A -85,B 0,C 180,E1 -21281.6,E2 -21281.6} C_VEL
LIN {X 0,Y 206.741,Z 380.728,A -85,B 0,C 180,E1 -21285.552,E2 -21285.552} C_VEL
LIN {X 0,Y 206.741,Z 380.731,A -85,B 0,C 180,E1 -21289.771,E2 -21289.771} C_VEL
LIN {X 0,Y 206.959,Z 380.846,A -85,B 0,C 180,E1 -21294.966,E2 -21294.966} C_VEL
LIN {X 0,Y 210.143,Z 396.651,A -85,B 0,C 180,E1 -21301.043,E2 -21301.043} C_VEL
LIN {X 0,Y 210.416,Z 398.169,A -85,B 0,C 180,E1 -21301.605,E2 -21301.605} C_VEL
LIN {X 0,Y 210.058,Z 400.383,A -85,B 0,C 180,E1 -21302.411,E2 -21302.411} C_VEL
LIN {X 0,Y 210.203,Z 417.537,A -85,B 0,C 180,E1 -21303.467,E2 -21303.467} C_VEL
LIN {X 0,Y 212.231,Z 446.458,A -85,B 0,C 180,E1 -21305.249,E2 -21305.249} C_VEL
LIN {X 0,Y 213.143,Z 458.524,A -85,B 0,C 180,E1 -21305.985,E2 -21305.985} C_VEL
LIN {X 0,Y 212.831,Z 465.826,A -85,B 0,C 180,E1 -21306.415,E2 -21306.415} C_VEL
LIN {X 0,Y 211.868,Z 471.539,A -85,B 0,C 180,E1 -21306.743,E2 -21306.743} C_VEL
LIN {X 0,Y 205.275,Z 489.866,A -85,B 0,C 180,E1 -21307.812,E2 -21307.812} C_VEL
LIN {X 0,Y 204.485,Z 495.574,A -85,B 0,C 180,E1 -21308.171,E2 -21308.171} C_VEL
LIN {X 0,Y 203.796,Z 513.848,A -85,B 0,C 180,E1 -21309.443,E2 -21309.443} C_VEL
LIN {X 0,Y 202.9,Z 527.199,A -85,B 0,C 180,E1 -21310.791,E2 -21310.791} C_VEL
LIN {X 0,Y 201.878,Z 540.224,A -85,B 0,C 180,E1 -21312.529,E2 -21312.529} C_VEL
LIN {X 0,Y 200.918,Z 553.313,A -85,B 0,C 180,E1 -21314.793,E2 -21314.793} C_VEL
LIN {X 0,Y 200.114,Z 564.766,A -85,B 0,C 180,E1 -21317.323,E2 -21317.323} C_VEL
LIN {X 0,Y 199.673,Z 574.15,A -85,B 0,C 180,E1 -21319.866,E2 -21319.866} C_VEL
LIN {X 0,Y 199.476,Z 583.176,A -85,B 0,C 180,E1 -21322.919,E2 -21322.919} C_VEL
LIN {X 0,Y 199.564,Z 590.343,A -85,B 0,C 180,E1 -21325.963,E2 -21325.963} C_VEL
LIN {X 0,Y 199.573,Z 595.875,A -85,B 0,C 180,E1 -21328.993,E2 -21328.993} C_VEL
LIN {X 0,Y 199.378,Z 598.697,A -85,B 0,C 180,E1 -21331.012,E2 -21331.012} C_VEL
LIN {X 0,Y 198.607,Z 601.877,A -85,B 0,C 180,E1 -21334.061,E2 -21334.061} C_VEL
LIN {X 0,Y 198.221,Z 603.922,A -85,B 0,C 180,E1 -21336.899,E2 -21336.899} C_VEL
LIN {X 0,Y 198.209,Z 605.359,A -85,B 0,C 180,E1 -21340.214,E2 -21340.214} C_VEL
LIN {X 0,Y 199.277,Z 605.896,A -85,B 0,C 180,E1 -21344.295,E2 -21344.295} C_VEL
LIN {X 0,Y 201.736,Z 605.075,A -85,B 0,C 180,E1 -21348.275,E2 -21348.275} C_VEL
LIN {X 0,Y 205.287,Z 602.853,A -85,B 0,C 180,E1 -21352.125,E2 -21352.125} C_VEL
LIN {X 0,Y 207.552,Z 601.23,A -85,B 0,C 180,E1 -21353.977,E2 -21353.977} C_VEL
LIN {X 0,Y 213.017,Z 596.926,A -85,B 0,C 180,E1 -21357.512,E2 -21357.512} C_VEL
LIN {X 0,Y 219.718,Z 591.089,A -85,B 0,C 180,E1 -21360.785,E2 -21360.785} C_VEL
LIN {X 0,Y 227.348,Z 583.521,A -85,B 0,C 180,E1 -21363.812,E2 -21363.812} C_VEL
LIN {X 0,Y 234.87,Z 575.309,A -85,B 0,C 180,E1 -21366.229,E2 -21366.229} C_VEL
LIN {X 0,Y 242.937,Z 565.378,A -85,B 0,C 180,E1 -21368.436,E2 -21368.436} C_VEL
LIN {X 0,Y 250.708,Z 554.829,A -85,B 0,C 180,E1 -21370.149,E2 -21370.149} C_VEL
LIN {X 0,Y 258.181,Z 543.216,A -85,B 0,C 180,E1 -21371.571,E2 -21371.571} C_VEL
LIN {X 0,Y 265.311,Z 530.468,A -85,B 0,C 180,E1 -21372.752,E2 -21372.752} C_VEL
LIN {X 0,Y 271.941,Z 516.296,A -85,B 0,C 180,E1 -21373.738,E2 -21373.738} C_VEL
LIN {X 0,Y 277.824,Z 500.695,A -85,B 0,C 180,E1 -21374.562,E2 -21374.562} C_VEL
LIN {X 0,Y 281.796,Z 487.165,A -85,B 0,C 180,E1 -21375.2,E2 -21375.2} C_VEL
LIN {X 0,Y 281.944,Z 486.418,A -85,B 0,C 180,E1 -21376.138,E2 -21376.138} C_VEL
LIN {X 0,Y 277.685,Z 500.387,A -85,B 0,C 180,E1 -21376.894,E2 -21376.894} C_VEL
LIN {X 0,Y 273.09,Z 512.284,A -85,B 0,C 180,E1 -21377.752,E2 -21377.752} C_VEL
LIN {X 0,Y 267.932,Z 523.308,A -85,B 0,C 180,E1 -21378.773,E2 -21378.773} C_VEL
LIN {X 0,Y 261.089,Z 535.609,A -85,B 0,C 180,E1 -21380.26,E2 -21380.26} C_VEL
LIN {X 0,Y 255.022,Z 544.871,A -85,B 0,C 180,E1 -21381.679,E2 -21381.679} C_VEL
LIN {X 0,Y 248.074,Z 554.135,A -85,B 0,C 180,E1 -21383.492,E2 -21383.492} C_VEL
LIN {X 0,Y 241.455,Z 561.826,A -85,B 0,C 180,E1 -21385.418,E2 -21385.418} C_VEL
LIN {X 0,Y 235.144,Z 568.191,A -85,B 0,C 180,E1 -21387.453,E2 -21387.453} C_VEL
LIN {X 0,Y 229.341,Z 573.342,A -85,B 0,C 180,E1 -21389.626,E2 -21389.626} C_VEL
LIN {X 0,Y 223.931,Z 577.48,A -85,B 0,C 180,E1 -21391.915,E2 -21391.915} C_VEL
LIN {X 0,Y 217.515,Z 581.472,A -85,B 0,C 180,E1 -21395.163,E2 -21395.163} C_VEL
LIN {X 0,Y 214.557,Z 582.921,A -85,B 0,C 180,E1 -21396.854,E2 -21396.854} C_VEL
LIN {X 0,Y 209.424,Z 584.599,A -85,B 0,C 180,E1 -21400.391,E2 -21400.391} C_VEL
LIN {X 0,Y 205.198,Z 584.795,A -85,B 0,C 180,E1 -21404.097,E2 -21404.097} C_VEL
LIN {X 0,Y 201.903,Z 583.52,A -85,B 0,C 180,E1 -21407.945,E2 -21407.945} C_VEL
LIN {X 0,Y 199.873,Z 580.673,A -85,B 0,C 180,E1 -21411.914,E2 -21411.914} C_VEL
LIN {X 0,Y 198.821,Z 577.526,A -85,B 0,C 180,E1 -21414.93,E2 -21414.93} C_VEL
LIN {X 0,Y 198.071,Z 573.401,A -85,B 0,C 180,E1 -21417.966,E2 -21417.966} C_VEL
LIN {X 0,Y 197.869,Z 568.193,A -85,B 0,C 180,E1 -21421.017,E2 -21421.017} C_VEL
LIN {X 0,Y 198.092,Z 561.773,A -85,B 0,C 180,E1 -21424.069,E2 -21424.069} C_VEL
LIN {X 0,Y 198.468,Z 552.921,A -85,B 0,C 180,E1 -21427.454,E2 -21427.454} C_VEL
LIN {X 0,Y 198.995,Z 544.116,A -85,B 0,C 180,E1 -21430.171,E2 -21430.171} C_VEL
LIN {X 0,Y 199.851,Z 533.112,A -85,B 0,C 180,E1 -21432.955,E2 -21432.955} C_VEL
LIN {X 0,Y 200.822,Z 522.13,A -85,B 0,C 180,E1 -21435.217,E2 -21435.217} C_VEL
LIN {X 0,Y 201.94,Z 508.406,A -85,B 0,C 180,E1 -21437.468,E2 -21437.468} C_VEL
LIN {X 0,Y 202.915,Z 493.396,A -85,B 0,C 180,E1 -21439.341,E2 -21439.341} C_VEL
LIN {X 0,Y 203.871,Z 478.624,A -85,B 0,C 180,E1 -21440.68,E2 -21440.68} C_VEL
LIN {X 0,Y 206.97,Z 407.999,A -85,B 0,C 180,E1 -21445.029,E2 -21445.029} C_VEL
LIN {X 0,Y 199.776,Z 381.599,A -85,B 0,C 180,E1 -21446.969,E2 -21446.969} C_VEL
LIN {X 0,Y 199.685,Z 381.608,A -85,B 0,C 180,E1 -21452.358,E2 -21452.358} C_VEL
LIN {X 0,Y 199.629,Z 381.618,A -85,B 0,C 180,E1 -21456.762,E2 -21456.762} C_VEL
LIN {X 0,Y 199.614,Z 381.618,A -85,B 0,C 180,E1 -21459.327,E2 -21459.327} C_VEL
LIN {X 0,Y 199.579,Z 381.622,A -85,B 0,C 180,E1 -21462.309,E2 -21462.309} C_VEL
LIN {X 0,Y 199.585,Z 381.622,A -85,B 0,C 180,E1 -21465.227,E2 -21465.227} C_VEL
LIN {X 0,Y 199.643,Z 381.613,A -85,B 0,C 180,E1 -21470.677,E2 -21470.677} C_VEL
LIN {X 0,Y 199.639,Z 381.616,A -85,B 0,C 180,E1 -21475.716,E2 -21475.716} C_VEL
LIN {X 0,Y 199.708,Z 381.606,A -85,B 0,C 180,E1 -21478.136,E2 -21478.136} C_VEL
LIN {X 0,Y 199.691,Z 381.609,A -85,B 0,C 180,E1 -21482.77,E2 -21482.77} C_VEL
LIN {X 0,Y 199.742,Z 381.6,A -85,B 0,C 180,E1 -21487.227,E2 -21487.227} C_VEL
LIN {X 0,Y 199.8,Z 381.596,A -85,B 0,C 180,E1 -21491.755,E2 -21491.755} C_VEL
LIN {X 0,Y 199.839,Z 381.59,A -85,B 0,C 180,E1 -21495.746,E2 -21495.746} C_VEL
LIN {X 0,Y 200.025,Z 381.569,A -85,B 0,C 180,E1 -21499.88,E2 -21499.88} C_VEL
LIN {X 0,Y 200.026,Z 381.568,A -85,B 0,C 180,E1 -21503.947,E2 -21503.947} C_VEL
LIN {X 0,Y 200.324,Z 381.531,A -85,B 0,C 180,E1 -21507.987,E2 -21507.987} C_VEL
LIN {X 0,Y 200.484,Z 381.514,A -85,B 0,C 180,E1 -21509.998,E2 -21509.998} C_VEL
LIN {X 0,Y 200.035,Z 381.565,A -85,B 0,C 180,E1 -21514.027,E2 -21514.027} C_VEL
LIN {X 0,Y 200.133,Z 381.557,A -85,B 0,C 180,E1 -21518.072,E2 -21518.072} C_VEL
LIN {X 0,Y 199.914,Z 381.579,A -85,B 0,C 180,E1 -21522.174,E2 -21522.174} C_VEL
LIN {X 0,Y 199.804,Z 381.596,A -85,B 0,C 180,E1 -21526.341,E2 -21526.341} C_VEL
LIN {X 0,Y 199.698,Z 381.606,A -85,B 0,C 180,E1 -21530.603,E2 -21530.603} C_VEL
LIN {X 0,Y 199.67,Z 381.611,A -85,B 0,C 180,E1 -21534.982,E2 -21534.982} C_VEL
LIN {X 0,Y 199.671,Z 381.612,A -85,B 0,C 180,E1 -21539.52,E2 -21539.52} C_VEL
LIN {X 0,Y 199.66,Z 381.612,A -85,B 0,C 180,E1 -21542.35,E2 -21542.35} C_VEL
LIN {X 0,Y 199.649,Z 381.613,A -85,B 0,C 180,E1 -21546.754,E2 -21546.754} C_VEL
LIN {X 0,Y 199.696,Z 381.606,A -85,B 0,C 180,E1 -21549.304,E2 -21549.304} C_VEL
LIN {X 0,Y 199.684,Z 381.61,A -85,B 0,C 180,E1 -21552.345,E2 -21552.345} C_VEL
LIN {X 0,Y 199.688,Z 381.61,A -85,B 0,C 180,E1 -21555.26,E2 -21555.26} C_VEL
LIN {X 0,Y 199.692,Z 381.607,A -85,B 0,C 180,E1 -21558.034,E2 -21558.034} C_VEL
LIN {X 0,Y 199.696,Z 381.607,A -85,B 0,C 180,E1 -21560.734,E2 -21560.734} C_VEL
LIN {X 0,Y 199.628,Z 381.616,A -85,B 0,C 180,E1 -21565.717,E2 -21565.717} C_VEL
LIN {X 0,Y 199.697,Z 381.607,A -85,B 0,C 180,E1 -21568.136,E2 -21568.136} C_VEL
LIN {X 0,Y 199.679,Z 381.61,A -85,B 0,C 180,E1 -21572.771,E2 -21572.771} C_VEL
LIN {X 0,Y 199.73,Z 381.602,A -85,B 0,C 180,E1 -21577.228,E2 -21577.228} C_VEL
LIN {X 0,Y 199.788,Z 381.598,A -85,B 0,C 180,E1 -21581.757,E2 -21581.757} C_VEL
LIN {X 0,Y 199.839,Z 381.591,A -85,B 0,C 180,E1 -21585.749,E2 -21585.749} C_VEL
LIN {X 0,Y 200.067,Z 381.563,A -85,B 0,C 180,E1 -21589.884,E2 -21589.884} C_VEL
LIN {X 0,Y 200.124,Z 381.553,A -85,B 0,C 180,E1 -21591.925,E2 -21591.925} C_VEL
LIN {X 0,Y 200.316,Z 381.532,A -85,B 0,C 180,E1 -21597.99,E2 -21597.99} C_VEL
LIN {X 0,Y 200.475,Z 381.51,A -85,B 0,C 180,E1 -21600,E2 -21600} C_VEL
LIN {X 0,Y 200.027,Z 381.567,A -85,B 0,C 180,E1 -21604.03,E2 -21604.03} C_VEL
LIN {X 0,Y 200.124,Z 381.555,A -85,B 0,C 180,E1 -21608.075,E2 -21608.075} C_VEL
LIN {X 0,Y 199.907,Z 381.58,A -85,B 0,C 180,E1 -21612.178,E2 -21612.178} C_VEL
LIN {X 0,Y 199.798,Z 381.595,A -85,B 0,C 180,E1 -21616.344,E2 -21616.344} C_VEL
LIN {X 0,Y 199.816,Z 381.591,A -85,B 0,C 180,E1 -21618.455,E2 -21618.455} C_VEL
LIN {X 0,Y 199.729,Z 381.605,A -85,B 0,C 180,E1 -21623.818,E2 -21623.818} C_VEL
LIN {X 0,Y 199.701,Z 381.603,A -85,B 0,C 180,E1 -21628.386,E2 -21628.386} C_VEL
LIN {X 0,Y 199.651,Z 381.614,A -85,B 0,C 180,E1 -21632.351,E2 -21632.351} C_VEL
LIN {X 0,Y 199.658,Z 381.611,A -85,B 0,C 180,E1 -21636.756,E2 -21636.756} C_VEL
LIN {X 0,Y 199.718,Z 381.606,A -85,B 0,C 180,E1 -21639.303,E2 -21639.303} C_VEL
LIN {X 0,Y 199.697,Z 381.608,A -85,B 0,C 180,E1 -21642.353,E2 -21642.353} C_VEL
LIN {X 0,Y 199.689,Z 381.608,A -85,B 0,C 180,E1 -21645.264,E2 -21645.264} C_VEL
LIN {X 0,Y 199.687,Z 381.608,A -85,B 0,C 180,E1 -21648.036,E2 -21648.036} C_VEL
LIN {X 0,Y 199.743,Z 381.602,A -85,B 0,C 180,E1 -21653.266,E2 -21653.266} C_VEL
LIN {X 0,Y 199.899,Z 381.759,A -85,B 0,C 180,E1 -21654.945,E2 -21654.945} C_VEL
LIN {X 0,Y 203.016,Z 396.987,A -85,B 0,C 180,E1 -21661.013,E2 -21661.013} C_VEL
LIN {X 0,Y 203.291,Z 398.571,A -85,B 0,C 180,E1 -21661.62,E2 -21661.62} C_VEL
LIN {X 0,Y 203.048,Z 399.963,A -85,B 0,C 180,E1 -21662.146,E2 -21662.146} C_VEL
LIN {X 0,Y 203.174,Z 418.157,A -85,B 0,C 180,E1 -21663.279,E2 -21663.279} C_VEL
LIN {X 0,Y 205.221,Z 447.454,A -85,B 0,C 180,E1 -21665.162,E2 -21665.162} C_VEL
LIN {X 0,Y 206.083,Z 458.19,A -85,B 0,C 180,E1 -21665.846,E2 -21665.846} C_VEL
LIN {X 0,Y 204.485,Z 495.574,A -85,B 0,C 180,E1 -21668.171,E2 -21668.171} C_VEL
LIN {X 0,Y 203.664,Z 501.279,A -85,B 0,C 180,E1 -21668.533,E2 -21668.533} C_VEL
LIN {X 0,Y 200.377,Z 510.358,A -85,B 0,C 180,E1 -21669.194,E2 -21669.194} C_VEL
LIN {X 0,Y 196.987,Z 519.27,A -85,B 0,C 180,E1 -21670.039,E2 -21670.039} C_VEL
LIN {X 0,Y 195.952,Z 524.725,A -85,B 0,C 180,E1 -21670.661,E2 -21670.661} C_VEL
LIN {X 0,Y 194.95,Z 537.879,A -85,B 0,C 180,E1 -21672.43,E2 -21672.43} C_VEL
LIN {X 0,Y 194.09,Z 549.958,A -85,B 0,C 180,E1 -21674.514,E2 -21674.514} C_VEL
LIN {X 0,Y 193.268,Z 560.852,A -85,B 0,C 180,E1 -21676.866,E2 -21676.866} C_VEL
LIN {X 0,Y 192.797,Z 570.761,A -85,B 0,C 180,E1 -21679.501,E2 -21679.501} C_VEL
LIN {X 0,Y 192.573,Z 578.875,A -85,B 0,C 180,E1 -21682.136,E2 -21682.136} C_VEL
LIN {X 0,Y 192.629,Z 585.59,A -85,B 0,C 180,E1 -21684.769,E2 -21684.769} C_VEL
LIN {X 0,Y 192.726,Z 591.988,A -85,B 0,C 180,E1 -21687.913,E2 -21687.913} C_VEL
LIN {X 0,Y 192.691,Z 595.408,A -85,B 0,C 180,E1 -21690.002,E2 -21690.002} C_VEL
LIN {X 0,Y 192.26,Z 598.067,A -85,B 0,C 180,E1 -21692.097,E2 -21692.097} C_VEL
LIN {X 0,Y 191.729,Z 600.211,A -85,B 0,C 180,E1 -21694.207,E2 -21694.207} C_VEL
LIN {X 0,Y 191.194,Z 603.247,A -85,B 0,C 180,E1 -21698.457,E2 -21698.457} C_VEL
LIN {X 0,Y 191.681,Z 604.79,A -85,B 0,C 180,E1 -21702.711,E2 -21702.711} C_VEL
LIN {X 0,Y 193.593,Z 604.974,A -85,B 0,C 180,E1 -21706.886,E2 -21706.886} C_VEL
LIN {X 0,Y 196.752,Z 603.826,A -85,B 0,C 180,E1 -21710.931,E2 -21710.931} C_VEL
LIN {X 0,Y 201.086,Z 601.358,A -85,B 0,C 180,E1 -21714.799,E2 -21714.799} C_VEL
LIN {X 0,Y 206.78,Z 597.542,A -85,B 0,C 180,E1 -21718.416,E2 -21718.416} C_VEL
LIN {X 0,Y 213.733,Z 592.217,A -85,B 0,C 180,E1 -21721.746,E2 -21721.746} C_VEL
LIN {X 0,Y 221.629,Z 585.309,A -85,B 0,C 180,E1 -21724.808,E2 -21724.808} C_VEL
LIN {X 0,Y 229.334,Z 577.785,A -85,B 0,C 180,E1 -21727.249,E2 -21727.249} C_VEL
LIN {X 0,Y 237.656,Z 568.652,A -85,B 0,C 180,E1 -21729.454,E2 -21729.454} C_VEL
LIN {X 0,Y 245.552,Z 559.045,A -85,B 0,C 180,E1 -21731.171,E2 -21731.171} C_VEL
LIN {X 0,Y 253.21,Z 548.555,A -85,B 0,C 180,E1 -21732.576,E2 -21732.576} C_VEL
LIN {X 0,Y 260.427,Z 537.199,A -85,B 0,C 180,E1 -21733.753,E2 -21733.753} C_VEL
LIN {X 0,Y 267.739,Z 523.823,A -85,B 0,C 180,E1 -21734.788,E2 -21734.788} C_VEL
LIN {X 0,Y 274.222,Z 509.495,A -85,B 0,C 180,E1 -21735.625,E2 -21735.625} C_VEL
LIN {X 0,Y 274.888,Z 507.783,A -85,B 0,C 180,E1 -21735.716,E2 -21735.716} C_VEL
LIN {X 0,Y 274.41,Z 508.953,A -85,B 0,C 180,E1 -21735.935,E2 -21735.935} C_VEL
LIN {X 0,Y 268.801,Z 520.979,A -85,B 0,C 180,E1 -21736.916,E2 -21736.916} C_VEL
LIN {X 0,Y 262.222,Z 532.77,A -85,B 0,C 180,E1 -21738.187,E2 -21738.187} C_VEL
LIN {X 0,Y 255.162,Z 543.435,A -85,B 0,C 180,E1 -21739.664,E2 -21739.664} C_VEL
LIN {X 0,Y 247.779,Z 553.028,A -85,B 0,C 180,E1 -21741.39,E2 -21741.39} C_VEL
LIN {X 0,Y 239.537,Z 562.19,A -85,B 0,C 180,E1 -21743.549,E2 -21743.549} C_VEL
LIN {X 0,Y 231.765,Z 569.518,A -85,B 0,C 180,E1 -21745.875,E2 -21745.875} C_VEL
LIN {X 0,Y 225.559,Z 574.558,A -85,B 0,C 180,E1 -21748.015,E2 -21748.015} C_VEL
LIN {X 0,Y 217.971,Z 579.716,A -85,B 0,C 180,E1 -21751.076,E2 -21751.076} C_VEL
LIN {X 0,Y 214.515,Z 581.664,A -85,B 0,C 180,E1 -21752.698,E2 -21752.698} C_VEL
LIN {X 0,Y 208.191,Z 584.386,A -85,B 0,C 180,E1 -21756.103,E2 -21756.103} C_VEL
LIN {X 0,Y 202.835,Z 585.645,A -85,B 0,C 180,E1 -21759.727,E2 -21759.727} C_VEL
LIN {X 0,Y 198.427,Z 585.414,A -85,B 0,C 180,E1 -21763.54,E2 -21763.54} C_VEL
LIN {X 0,Y 194.969,Z 583.709,A -85,B 0,C 180,E1 -21767.509,E2 -21767.509} C_VEL
LIN {X 0,Y 192.869,Z 580.528,A -85,B 0,C 180,E1 -21771.619,E2 -21771.619} C_VEL
LIN {X 0,Y 191.77,Z 577.076,A -85,B 0,C 180,E1 -21774.743,E2 -21774.743} C_VEL
LIN {X 0,Y 191.008,Z 572.632,A -85,B 0,C 180,E1 -21777.891,E2 -21777.891} C_VEL
LIN {X 0,Y 190.854,Z 566.079,A -85,B 0,C 180,E1 -21781.582,E2 -21781.582} C_VEL
LIN {X 0,Y 191.094,Z 559.045,A -85,B 0,C 180,E1 -21784.745,E2 -21784.745} C_VEL
LIN {X 0,Y 191.56,Z 549.92,A -85,B 0,C 180,E1 -21788.081,E2 -21788.081} C_VEL
LIN {X 0,Y 192.252,Z 539.766,A -85,B 0,C 180,E1 -21791.065,E2 -21791.065} C_VEL
LIN {X 0,Y 193.11,Z 528.893,A -85,B 0,C 180,E1 -21793.683,E2 -21793.683} C_VEL
LIN {X 0,Y 194.123,Z 516.782,A -85,B 0,C 180,E1 -21796.025,E2 -21796.025} C_VEL
LIN {X 0,Y 195.059,Z 505.224,A -85,B 0,C 180,E1 -21797.834,E2 -21797.834} C_VEL
LIN {X 0,Y 195.972,Z 491.536,A -85,B 0,C 180,E1 -21799.51,E2 -21799.51} C_VEL
LIN {X 0,Y 196.794,Z 477.46,A -85,B 0,C 180,E1 -21800.787,E2 -21800.787} C_VEL
LIN {X 0,Y 199.81,Z 408.853,A -85,B 0,C 180,E1 -21805.2,E2 -21805.2} C_VEL
LIN {X 0,Y 192.723,Z 382.477,A -85,B 0,C 180,E1 -21807.191,E2 -21807.191} C_VEL
LIN {X 0,Y 192.617,Z 382.486,A -85,B 0,C 180,E1 -21812.941,E2 -21812.941} C_VEL
LIN {X 0,Y 192.592,Z 382.495,A -85,B 0,C 180,E1 -21816.597,E2 -21816.597} C_VEL
LIN {X 0,Y 192.519,Z 382.498,A -85,B 0,C 180,E1 -21821.079,E2 -21821.079} C_VEL
LIN {X 0,Y 192.497,Z 382.508,A -85,B 0,C 180,E1 -21826.075,E2 -21826.075} C_VEL
LIN {X 0,Y 192.544,Z 382.498,A -85,B 0,C 180,E1 -21830.042,E2 -21830.042} C_VEL
LIN {X 0,Y 192.603,Z 382.495,A -85,B 0,C 180,E1 -21834.277,E2 -21834.277} C_VEL
LIN {X 0,Y 192.612,Z 382.486,A -85,B 0,C 180,E1 -21839.278,E2 -21839.278} C_VEL
LIN {X 0,Y 192.669,Z 382.483,A -85,B 0,C 180,E1 -21841.69,E2 -21841.69} C_VEL
LIN {X 0,Y 192.71,Z 382.478,A -85,B 0,C 180,E1 -21846.347,E2 -21846.347} C_VEL
LIN {X 0,Y 192.735,Z 382.475,A -85,B 0,C 180,E1 -21851.455,E2 -21851.455} C_VEL
LIN {X 0,Y 192.767,Z 382.47,A -85,B 0,C 180,E1 -21855.212,E2 -21855.212} C_VEL
LIN {X 0,Y 192.947,Z 382.449,A -85,B 0,C 180,E1 -21859.564,E2 -21859.564} C_VEL
LIN {X 0,Y 192.988,Z 382.445,A -85,B 0,C 180,E1 -21863.726,E2 -21863.726} C_VEL
LIN {X 0,Y 193.266,Z 382.41,A -85,B 0,C 180,E1 -21867.914,E2 -21867.914} C_VEL
LIN {X 0,Y 193.448,Z 382.39,A -85,B 0,C 180,E1 -21869.998,E2 -21869.998} C_VEL
LIN {X 0,Y 192.982,Z 382.442,A -85,B 0,C 180,E1 -21874.174,E2 -21874.174} C_VEL
LIN {X 0,Y 193.079,Z 382.434,A -85,B 0,C 180,E1 -21878.369,E2 -21878.369} C_VEL
LIN {X 0,Y 192.853,Z 382.457,A -85,B 0,C 180,E1 -21882.627,E2 -21882.627} C_VEL
LIN {X 0,Y 192.757,Z 382.473,A -85,B 0,C 180,E1 -21886.956,E2 -21886.956} C_VEL
LIN {X 0,Y 192.635,Z 382.486,A -85,B 0,C 180,E1 -21891.395,E2 -21891.395} C_VEL
LIN {X 0,Y 192.661,Z 382.486,A -85,B 0,C 180,E1 -21894.222,E2 -21894.222} C_VEL
LIN {X 0,Y 192.646,Z 382.485,A -85,B 0,C 180,E1 -21898.89,E2 -21898.89} C_VEL
LIN {X 0,Y 192.596,Z 382.492,A -85,B 0,C 180,E1 -21903.183,E2 -21903.183} C_VEL
LIN {X 0,Y 192.608,Z 382.488,A -85,B 0,C 180,E1 -21908.335,E2 -21908.335} C_VEL
LIN {X 0,Y 192.622,Z 382.49,A -85,B 0,C 180,E1 -21913.137,E2 -21913.137} C_VEL
LIN {X 0,Y 192.627,Z 382.487,A -85,B 0,C 180,E1 -21916.857,E2 -21916.857} C_VEL
LIN {X 0,Y 192.606,Z 382.494,A -85,B 0,C 180,E1 -21921.661,E2 -21921.661} C_VEL
LIN {X 0,Y 192.593,Z 382.489,A -85,B 0,C 180,E1 -21926.813,E2 -21926.813} C_VEL
LIN {X 0,Y 192.657,Z 382.488,A -85,B 0,C 180,E1 -21931.691,E2 -21931.691} C_VEL
LIN {X 0,Y 192.698,Z 382.477,A -85,B 0,C 180,E1 -21936.348,E2 -21936.348} C_VEL
LIN {X 0,Y 192.724,Z 382.479,A -85,B 0,C 180,E1 -21941.457,E2 -21941.457} C_VEL
LIN {X 0,Y 192.763,Z 382.468,A -85,B 0,C 180,E1 -21945.214,E2 -21945.214} C_VEL
LIN {X 0,Y 193.012,Z 382.444,A -85,B 0,C 180,E1 -21949.51,E2 -21949.51} C_VEL
LIN {X 0,Y 192.997,Z 382.441,A -85,B 0,C 180,E1 -21953.728,E2 -21953.728} C_VEL
LIN {X 0,Y 193.258,Z 382.411,A -85,B 0,C 180,E1 -21957.916,E2 -21957.916} C_VEL
LIN {X 0,Y 193.438,Z 382.387,A -85,B 0,C 180,E1 -21960,E2 -21960} C_VEL
LIN {X 0,Y 192.974,Z 382.445,A -85,B 0,C 180,E1 -21964.177,E2 -21964.177} C_VEL
LIN {X 0,Y 193.071,Z 382.433,A -85,B 0,C 180,E1 -21968.373,E2 -21968.373} C_VEL
LIN {X 0,Y 192.846,Z 382.46,A -85,B 0,C 180,E1 -21972.631,E2 -21972.631} C_VEL
LIN {X 0,Y 192.773,Z 382.468,A -85,B 0,C 180,E1 -21978.587,E2 -21978.587} C_VEL
LIN {X 0,Y 192.657,Z 382.485,A -85,B 0,C 180,E1 -21984.226,E2 -21984.226} C_VEL
LIN {X 0,Y 192.637,Z 382.484,A -85,B 0,C 180,E1 -21988.89,E2 -21988.89} C_VEL
LIN {X 0,Y 192.591,Z 382.496,A -85,B 0,C 180,E1 -21993.188,E2 -21993.188} C_VEL
LIN {X 0,Y 192.623,Z 382.486,A -85,B 0,C 180,E1 -21998.335,E2 -21998.335} C_VEL
LIN {X 0,Y 192.629,Z 382.491,A -85,B 0,C 180,E1 -22003.144,E2 -22003.144} C_VEL
LIN {X 0,Y 192.623,Z 382.486,A -85,B 0,C 180,E1 -22006.863,E2 -22006.863} C_VEL
LIN {X 0,Y 192.639,Z 382.488,A -85,B 0,C 180,E1 -22011.672,E2 -22011.672} C_VEL
LIN {X 0,Y 192.854,Z 382.545,A -85,B 0,C 180,E1 -22014.922,E2 -22014.922} C_VEL
LIN {X 0,Y 195.913,Z 397.402,A -85,B 0,C 180,E1 -22021.037,E2 -22021.037} C_VEL
LIN {X 0,Y 196.053,Z 399.488,A -85,B 0,C 180,E1 -22021.864,E2 -22021.864} C_VEL
LIN {X 0,Y 196.067,Z 417.036,A -85,B 0,C 180,E1 -22023.001,E2 -22023.001} C_VEL
LIN {X 0,Y 198.116,Z 447.858,A -85,B 0,C 180,E1 -22025.062,E2 -22025.062} C_VEL
LIN {X 0,Y 198.951,Z 459.43,A -85,B 0,C 180,E1 -22025.826,E2 -22025.826} C_VEL
LIN {X 0,Y 196.833,Z 510.17,A -85,B 0,C 180,E1 -22029.22,E2 -22029.22} C_VEL
LIN {X 0,Y 196.143,Z 522.19,A -85,B 0,C 180,E1 -22030.375,E2 -22030.375} C_VEL
LIN {X 0,Y 195.952,Z 524.725,A -85,B 0,C 180,E1 -22030.661,E2 -22030.661} C_VEL
LIN {X 0,Y 195.312,Z 528.302,A -85,B 0,C 180,E1 -22031.104,E2 -22031.104} C_VEL
LIN {X 0,Y 192.84,Z 535.042,A -85,B 0,C 180,E1 -22032.086,E2 -22032.086} C_VEL
LIN {X 0,Y 187.961,Z 546.189,A -85,B 0,C 180,E1 -22034.144,E2 -22034.144} C_VEL
LIN {X 0,Y 186.97,Z 551.026,A -85,B 0,C 180,E1 -22035.145,E2 -22035.145} C_VEL
LIN {X 0,Y 186.224,Z 562.194,A -85,B 0,C 180,E1 -22037.746,E2 -22037.746} C_VEL
LIN {X 0,Y 185.827,Z 572.598,A -85,B 0,C 180,E1 -22040.769,E2 -22040.769} C_VEL
LIN {X 0,Y 185.748,Z 581.549,A -85,B 0,C 180,E1 -22044.03,E2 -22044.03} C_VEL
LIN {X 0,Y 185.882,Z 587.6,A -85,B 0,C 180,E1 -22046.751,E2 -22046.751} C_VEL
LIN {X 0,Y 185.877,Z 593.263,A -85,B 0,C 180,E1 -22050.003,E2 -22050.003} C_VEL
LIN {X 0,Y 185.425,Z 596.139,A -85,B 0,C 180,E1 -22052.175,E2 -22052.175} C_VEL
LIN {X 0,Y 184.864,Z 598.458,A -85,B 0,C 180,E1 -22054.363,E2 -22054.363} C_VEL
LIN {X 0,Y 184.367,Z 601.068,A -85,B 0,C 180,E1 -22057.644,E2 -22057.644} C_VEL
LIN {X 0,Y 184.375,Z 602.866,A -85,B 0,C 180,E1 -22060.99,E2 -22060.99} C_VEL
LIN {X 0,Y 185.593,Z 604.059,A -85,B 0,C 180,E1 -22065.374,E2 -22065.374} C_VEL
LIN {X 0,Y 188.289,Z 603.968,A -85,B 0,C 180,E1 -22069.632,E2 -22069.632} C_VEL
LIN {X 0,Y 192.192,Z 602.573,A -85,B 0,C 180,E1 -22073.721,E2 -22073.721} C_VEL
LIN {X 0,Y 197.554,Z 599.884,A -85,B 0,C 180,E1 -22077.549,E2 -22077.549} C_VEL
LIN {X 0,Y 202.346,Z 596.96,A -85,B 0,C 180,E1 -22080.242,E2 -22080.242} C_VEL
LIN {X 0,Y 209.718,Z 591.85,A -85,B 0,C 180,E1 -22083.571,E2 -22083.571} C_VEL
LIN {X 0,Y 218.125,Z 585.131,A -85,B 0,C 180,E1 -22086.591,E2 -22086.591} C_VEL
LIN {X 0,Y 226.675,Z 577.463,A -85,B 0,C 180,E1 -22089.079,E2 -22089.079} C_VEL
LIN {X 0,Y 235.083,Z 568.975,A -85,B 0,C 180,E1 -22091.128,E2 -22091.128} C_VEL
LIN {X 0,Y 243.254,Z 559.727,A -85,B 0,C 180,E1 -22092.764,E2 -22092.764} C_VEL
LIN {X 0,Y 251.91,Z 548.638,A -85,B 0,C 180,E1 -22094.227,E2 -22094.227} C_VEL
LIN {X 0,Y 259.366,Z 537.642,A -85,B 0,C 180,E1 -22095.322,E2 -22095.322} C_VEL
LIN {X 0,Y 264.047,Z 529.838,A -85,B 0,C 180,E1 -22095.945,E2 -22095.945} C_VEL
LIN {X 0,Y 263.899,Z 530.022,A -85,B 0,C 180,E1 -22096.178,E2 -22096.178} C_VEL
LIN {X 0,Y 257.12,Z 540.314,A -85,B 0,C 180,E1 -22097.428,E2 -22097.428} C_VEL
LIN {X 0,Y 249.236,Z 550.554,A -85,B 0,C 180,E1 -22099.034,E2 -22099.034} C_VEL
LIN {X 0,Y 240.41,Z 560.303,A -85,B 0,C 180,E1 -22101.059,E2 -22101.059} C_VEL
LIN {X 0,Y 232.014,Z 568.112,A -85,B 0,C 180,E1 -22103.255,E2 -22103.255} C_VEL
LIN {X 0,Y 224.162,Z 574.358,A -85,B 0,C 180,E1 -22105.643,E2 -22105.643} C_VEL
LIN {X 0,Y 217.888,Z 578.561,A -85,B 0,C 180,E1 -22107.845,E2 -22107.845} C_VEL
LIN {X 0,Y 212.033,Z 581.833,A -85,B 0,C 180,E1 -22110.186,E2 -22110.186} C_VEL
LIN {X 0,Y 205.055,Z 584.842,A -85,B 0,C 180,E1 -22113.541,E2 -22113.541} C_VEL
LIN {X 0,Y 198.926,Z 586.341,A -85,B 0,C 180,E1 -22117.131,E2 -22117.131} C_VEL
LIN {X 0,Y 193.857,Z 586.413,A -85,B 0,C 180,E1 -22120.956,E2 -22120.956} C_VEL
LIN {X 0,Y 189.724,Z 585.056,A -85,B 0,C 180,E1 -22124.971,E2 -22124.971} C_VEL
LIN {X 0,Y 186.785,Z 582.183,A -85,B 0,C 180,E1 -22129.156,E2 -22129.156} C_VEL
LIN {X 0,Y 185.097,Z 577.827,A -85,B 0,C 180,E1 -22133.459,E2 -22133.459} C_VEL
LIN {X 0,Y 184.164,Z 573.41,A -85,B 0,C 180,E1 -22136.718,E2 -22136.718} C_VEL
LIN {X 0,Y 183.813,Z 566.921,A -85,B 0,C 180,E1 -22140.547,E2 -22140.547} C_VEL
LIN {X 0,Y 184.043,Z 559.991,A -85,B 0,C 180,E1 -22143.832,E2 -22143.832} C_VEL
LIN {X 0,Y 184.424,Z 550.982,A -85,B 0,C 180,E1 -22147.292,E2 -22147.292} C_VEL
LIN {X 0,Y 185.068,Z 541.015,A -85,B 0,C 180,E1 -22150.392,E2 -22150.392} C_VEL
LIN {X 0,Y 185.974,Z 529.127,A -85,B 0,C 180,E1 -22153.383,E2 -22153.383} C_VEL
LIN {X 0,Y 186.991,Z 517.023,A -85,B 0,C 180,E1 -22155.812,E2 -22155.812} C_VEL
LIN {X 0,Y 187.923,Z 505.495,A -85,B 0,C 180,E1 -22157.689,E2 -22157.689} C_VEL
LIN {X 0,Y 188.832,Z 491.778,A -85,B 0,C 180,E1 -22159.429,E2 -22159.429} C_VEL
LIN {X 0,Y 189.706,Z 477.757,A -85,B 0,C 180,E1 -22160.748,E2 -22160.748} C_VEL
LIN {X 0,Y 192.676,Z 409.821,A -85,B 0,C 180,E1 -22165.339,E2 -22165.339} C_VEL
LIN {X 0,Y 185.68,Z 383.354,A -85,B 0,C 180,E1 -22167.394,E2 -22167.394} C_VEL
LIN {X 0,Y 185.538,Z 383.368,A -85,B 0,C 180,E1 -22173.553,E2 -22173.553} C_VEL
LIN {X 0,Y 185.511,Z 383.375,A -85,B 0,C 180,E1 -22177.312,E2 -22177.312} C_VEL
LIN {X 0,Y 185.477,Z 383.376,A -85,B 0,C 180,E1 -22180.723,E2 -22180.723} C_VEL
LIN {X 0,Y 185.465,Z 383.383,A -85,B 0,C 180,E1 -22186.053,E2 -22186.053} C_VEL
LIN {X 0,Y 185.493,Z 383.376,A -85,B 0,C 180,E1 -22189.899,E2 -22189.899} C_VEL
LIN {X 0,Y 185.549,Z 383.371,A -85,B 0,C 180,E1 -22192.694,E2 -22192.694} C_VEL
LIN {X 0,Y 185.55,Z 383.37,A -85,B 0,C 180,E1 -22197.973,E2 -22197.973} C_VEL
LIN {X 0,Y 185.586,Z 383.366,A -85,B 0,C 180,E1 -22200.574,E2 -22200.574} C_VEL
LIN {X 0,Y 185.592,Z 383.365,A -85,B 0,C 180,E1 -22205.381,E2 -22205.381} C_VEL
LIN {X 0,Y 185.678,Z 383.354,A -85,B 0,C 180,E1 -22211.131,E2 -22211.131} C_VEL
LIN {X 0,Y 185.698,Z 383.351,A -85,B 0,C 180,E1 -22214.635,E2 -22214.635} C_VEL
LIN {X 0,Y 185.891,Z 383.327,A -85,B 0,C 180,E1 -22219.415,E2 -22219.415} C_VEL
LIN {X 0,Y 185.951,Z 383.32,A -85,B 0,C 180,E1 -22223.487,E2 -22223.487} C_VEL
LIN {X 0,Y 186.21,Z 383.288,A -85,B 0,C 180,E1 -22227.835,E2 -22227.835} C_VEL
LIN {X 0,Y 186.411,Z 383.266,A -85,B 0,C 180,E1 -22229.998,E2 -22229.998} C_VEL
LIN {X 0,Y 185.93,Z 383.32,A -85,B 0,C 180,E1 -22234.333,E2 -22234.333} C_VEL
LIN {X 0,Y 186.029,Z 383.311,A -85,B 0,C 180,E1 -22238.689,E2 -22238.689} C_VEL
LIN {X 0,Y 185.764,Z 383.339,A -85,B 0,C 180,E1 -22243.118,E2 -22243.118} C_VEL
LIN {X 0,Y 185.689,Z 383.355,A -85,B 0,C 180,E1 -22247.622,E2 -22247.622} C_VEL
LIN {X 0,Y 185.595,Z 383.363,A -85,B 0,C 180,E1 -22252.249,E2 -22252.249} C_VEL
LIN {X 0,Y 185.559,Z 383.369,A -85,B 0,C 180,E1 -22257.029,E2 -22257.029} C_VEL
LIN {X 0,Y 185.575,Z 383.367,A -85,B 0,C 180,E1 -22259.491,E2 -22259.491} C_VEL
LIN {X 0,Y 185.517,Z 383.375,A -85,B 0,C 180,E1 -22264.625,E2 -22264.625} C_VEL
LIN {X 0,Y 185.563,Z 383.369,A -85,B 0,C 180,E1 -22267.312,E2 -22267.312} C_VEL
LIN {X 0,Y 185.577,Z 383.364,A -85,B 0,C 180,E1 -22270.763,E2 -22270.763} C_VEL
LIN {X 0,Y 185.581,Z 383.366,A -85,B 0,C 180,E1 -22276.012,E2 -22276.012} C_VEL
LIN {X 0,Y 185.561,Z 383.37,A -85,B 0,C 180,E1 -22279.92,E2 -22279.92} C_VEL
LIN {X 0,Y 185.568,Z 383.368,A -85,B 0,C 180,E1 -22282.702,E2 -22282.702} C_VEL
LIN {X 0,Y 185.538,Z 383.371,A -85,B 0,C 180,E1 -22287.974,E2 -22287.974} C_VEL
LIN {X 0,Y 185.574,Z 383.367,A -85,B 0,C 180,E1 -22290.575,E2 -22290.575} C_VEL
LIN {X 0,Y 185.58,Z 383.365,A -85,B 0,C 180,E1 -22295.382,E2 -22295.382} C_VEL
LIN {X 0,Y 185.667,Z 383.357,A -85,B 0,C 180,E1 -22301.132,E2 -22301.132} C_VEL
LIN {X 0,Y 185.756,Z 383.344,A -85,B 0,C 180,E1 -22306.879,E2 -22306.879} C_VEL
LIN {X 0,Y 186.021,Z 383.313,A -85,B 0,C 180,E1 -22311.308,E2 -22311.308} C_VEL
LIN {X 0,Y 186.202,Z 383.291,A -85,B 0,C 180,E1 -22317.837,E2 -22317.837} C_VEL
LIN {X 0,Y 186.402,Z 383.263,A -85,B 0,C 180,E1 -22320,E2 -22320} C_VEL
LIN {X 0,Y 185.922,Z 383.323,A -85,B 0,C 180,E1 -22324.336,E2 -22324.336} C_VEL
LIN {X 0,Y 186.021,Z 383.311,A -85,B 0,C 180,E1 -22328.692,E2 -22328.692} C_VEL
LIN {X 0,Y 185.757,Z 383.344,A -85,B 0,C 180,E1 -22333.121,E2 -22333.121} C_VEL
LIN {X 0,Y 185.709,Z 383.35,A -85,B 0,C 180,E1 -22337.623,E2 -22337.623} C_VEL
LIN {X 0,Y 185.593,Z 383.364,A -85,B 0,C 180,E1 -22342.252,E2 -22342.252} C_VEL
LIN {X 0,Y 185.553,Z 383.37,A -85,B 0,C 180,E1 -22347.034,E2 -22347.034} C_VEL
LIN {X 0,Y 185.571,Z 383.367,A -85,B 0,C 180,E1 -22349.495,E2 -22349.495} C_VEL
LIN {X 0,Y 185.515,Z 383.375,A -85,B 0,C 180,E1 -22354.629,E2 -22354.629} C_VEL
LIN {X 0,Y 185.562,Z 383.367,A -85,B 0,C 180,E1 -22357.316,E2 -22357.316} C_VEL
LIN {X 0,Y 185.59,Z 383.366,A -85,B 0,C 180,E1 -22360.772,E2 -22360.772} C_VEL
LIN {X 0,Y 185.58,Z 383.362,A -85,B 0,C 180,E1 -22366.017,E2 -22366.017} C_VEL
LIN {X 0,Y 185.562,Z 383.369,A -85,B 0,C 180,E1 -22369.923,E2 -22369.923} C_VEL
LIN {X 0,Y 185.821,Z 383.407,A -85,B 0,C 180,E1 -22374.945,E2 -22374.945} C_VEL
LIN {X 0,Y 188.913,Z 398.469,A -85,B 0,C 180,E1 -22381.365,E2 -22381.365} C_VEL
LIN {X 0,Y 189.022,Z 399.281,A -85,B 0,C 180,E1 -22381.595,E2 -22381.595} C_VEL
LIN {X 0,Y 189.021,Z 417.412,A -85,B 0,C 180,E1 -22382.828,E2 -22382.828} C_VEL
LIN {X 0,Y 191.047,Z 448.203,A -85,B 0,C 180,E1 -22384.976,E2 -22384.976} C_VEL
LIN {X 0,Y 191.883,Z 459.294,A -85,B 0,C 180,E1 -22385.741,E2 -22385.741} C_VEL
LIN {X 0,Y 189.769,Z 509.456,A -85,B 0,C 180,E1 -22389.262,E2 -22389.262} C_VEL
LIN {X 0,Y 189.114,Z 521.45,A -85,B 0,C 180,E1 -22390.463,E2 -22390.463} C_VEL
LIN {X 0,Y 188.186,Z 533.603,A -85,B 0,C 180,E1 -22392.058,E2 -22392.058} C_VEL
LIN {X 0,Y 187.272,Z 546.347,A -85,B 0,C 180,E1 -22394.215,E2 -22394.215} C_VEL
LIN {X 0,Y 186.97,Z 551.026,A -85,B 0,C 180,E1 -22395.145,E2 -22395.145} C_VEL
LIN {X 0,Y 185.978,Z 555.726,A -85,B 0,C 180,E1 -22396.201,E2 -22396.201} C_VEL
LIN {X 0,Y 182.796,Z 562.716,A -85,B 0,C 180,E1 -22398.148,E2 -22398.148} C_VEL
LIN {X 0,Y 179.731,Z 569.19,A -85,B 0,C 180,E1 -22400.345,E2 -22400.345} C_VEL
LIN {X 0,Y 178.932,Z 573.096,A -85,B 0,C 180,E1 -22401.758,E2 -22401.758} C_VEL
